LIN {X 0,Y 234.227,Z 351.546,A -85,B 0,C 180,E1 9411.137,E2 9411.137} C_VEL
LIN {X 0,Y 232.184,Z 350.426,A -85,B 0,C 180,E1 9404.231,E2 9404.231} C_VEL
LIN {X 0,Y 231.874,Z 350.167,A -85,B 0,C 180,E1 9397.903,E2 9397.903} C_VEL
LIN {X 0,Y 232.888,Z 350.916,A -85,B 0,C 180,E1 9391.006,E2 9391.006} C_VEL
LIN {X 0,Y 234.314,Z 351.747,A -85,B 0,C 180,E1 9386.888,E2 9386.888} C_VEL
LIN {X 0,Y 236.206,Z 355.562,A -85,B 0,C 180,E1 9382.033,E2 9382.033} C_VEL
LIN {X 0,Y 238.881,Z 357.916,A -85,B 0,C 180,E1 9377.787,E2 9377.787} C_VEL
LIN {X 0,Y 241.494,Z 361.984,A -85,B 0,C 180,E1 9374.013,E2 9374.013} C_VEL
LIN {X 0,Y 243.571,Z 364.124,A -85,B 0,C 180,E1 9371.6,E2 9371.6} C_VEL
LIN {X 0,Y 247.204,Z 368.916,A -85,B 0,C 180,E1 9367.74,E2 9367.74} C_VEL
LIN {X 0,Y 252.401,Z 375.828,A -85,B 0,C 180,E1 9363.074,E2 9363.074} C_VEL
LIN {X 0,Y 256.798,Z 381.754,A -85,B 0,C 180,E1 9359.662,E2 9359.662} C_VEL
LIN {X 0,Y 261.47,Z 388.445,A -85,B 0,C 180,E1 9356.385,E2 9356.385} C_VEL
LIN {X 0,Y 268.294,Z 399.263,A -85,B 0,C 180,E1 9352.072,E2 9352.072} C_VEL
LIN {X 0,Y 276.387,Z 412.565,A -85,B 0,C 180,E1 9347.608,E2 9347.608} C_VEL
LIN {X 0,Y 284.443,Z 426.777,A -85,B 0,C 180,E1 9343.665,E2 9343.665} C_VEL
LIN {X 0,Y 289.912,Z 436.98,A -85,B 0,C 180,E1 9341.23,E2 9341.23} C_VEL
LIN {X 0,Y 275.033,Z 547.244,A -85,B 0,C 180,E1 9338.255,E2 9338.255} C_VEL
LIN {X 0,Y 273.431,Z 554.838,A -85,B 0,C 180,E1 9338.207,E2 9338.207} C_VEL
LIN {X 0,Y 266.861,Z 574.928,A -85,B 0,C 180,E1 9338.675,E2 9338.675} C_VEL
LIN {X 0,Y 265.438,Z 581.426,A -85,B 0,C 180,E1 9338.599,E2 9338.599} C_VEL
LIN {X 0,Y 260.934,Z 605.989,A -85,B 0,C 180,E1 9337.701,E2 9337.701} C_VEL
LIN {X 0,Y 255.076,Z 629.268,A -85,B 0,C 180,E1 9336.611,E2 9336.611} C_VEL
LIN {X 0,Y 248.158,Z 651.869,A -85,B 0,C 180,E1 9335.198,E2 9335.198} C_VEL
LIN {X 0,Y 240.392,Z 673.643,A -85,B 0,C 180,E1 9333.405,E2 9333.405} C_VEL
LIN {X 0,Y 231.725,Z 694.834,A -85,B 0,C 180,E1 9331.147,E2 9331.147} C_VEL
LIN {X 0,Y 223.215,Z 713.542,A -85,B 0,C 180,E1 9328.611,E2 9328.611} C_VEL
LIN {X 0,Y 213.828,Z 732.446,A -85,B 0,C 180,E1 9325.378,E2 9325.378} C_VEL
LIN {X 0,Y 204.768,Z 749.485,A -85,B 0,C 180,E1 9321.671,E2 9321.671} C_VEL
LIN {X 0,Y 196.426,Z 764.496,A -85,B 0,C 180,E1 9317.563,E2 9317.563} C_VEL
LIN {X 0,Y 188.528,Z 778.313,A -85,B 0,C 180,E1 9312.749,E2 9312.749} C_VEL
LIN {X 0,Y 181.922,Z 790.051,A -85,B 0,C 180,E1 9307.59,E2 9307.59} C_VEL
LIN {X 0,Y 176.376,Z 800.61,A -85,B 0,C 180,E1 9301.746,E2 9301.746} C_VEL
LIN {X 0,Y 172.499,Z 809.062,A -85,B 0,C 180,E1 9295.764,E2 9295.764} C_VEL
LIN {X 0,Y 170.003,Z 816.157,A -85,B 0,C 180,E1 9289.226,E2 9289.226} C_VEL
LIN {X 0,Y 169.005,Z 821.281,A -85,B 0,C 180,E1 9282.988,E2 9282.988} C_VEL
LIN {X 0,Y 168.985,Z 824.538,A -85,B 0,C 180,E1 9277.134,E2 9277.134} C_VEL
LIN {X 0,Y 169.187,Z 826.21,A -85,B 0,C 180,E1 9272.368,E2 9272.368} C_VEL
LIN {X 0,Y 169.127,Z 826.898,A -85,B 0,C 180,E1 9267.964,E2 9267.964} C_VEL
LIN {X 0,Y 168.776,Z 826.725,A -85,B 0,C 180,E1 9262.85,E2 9262.85} C_VEL
LIN {X 0,Y 168.789,Z 825.056,A -85,B 0,C 180,E1 9255.941,E2 9255.941} C_VEL
LIN {X 0,Y 170.369,Z 821.696,A -85,B 0,C 180,E1 9248.659,E2 9248.659} C_VEL
LIN {X 0,Y 174.906,Z 815.918,A -85,B 0,C 180,E1 9240.339,E2 9240.339} C_VEL
LIN {X 0,Y 182.577,Z 808.466,A -85,B 0,C 180,E1 9232.561,E2 9232.561} C_VEL
LIN {X 0,Y 195.682,Z 797.535,A -85,B 0,C 180,E1 9224.325,E2 9224.325} C_VEL
LIN {X 0,Y 212.712,Z 784.952,A -85,B 0,C 180,E1 9217.399,E2 9217.399} C_VEL
LIN {X 0,Y 222.74,Z 778.057,A -85,B 0,C 180,E1 9214.369,E2 9214.369} C_VEL
LIN {X 0,Y 204.082,Z 786.443,A -85,B 0,C 180,E1 9207.742,E2 9207.742} C_VEL
LIN {X 0,Y 189.979,Z 792.578,A -85,B 0,C 180,E1 9200.33,E2 9200.33} C_VEL
LIN {X 0,Y 180.154,Z 796.526,A -85,B 0,C 180,E1 9192.505,E2 9192.505} C_VEL
LIN {X 0,Y 173.807,Z 798.607,A -85,B 0,C 180,E1 9184.293,E2 9184.293} C_VEL
LIN {X 0,Y 170.626,Z 798.921,A -85,B 0,C 180,E1 9176.645,E2 9176.645} C_VEL
LIN {X 0,Y 169.369,Z 797.944,A -85,B 0,C 180,E1 9170.147,E2 9170.147} C_VEL
LIN {X 0,Y 168.986,Z 795.971,A -85,B 0,C 180,E1 9163.859,E2 9163.859} C_VEL
LIN {X 0,Y 169.098,Z 792.896,A -85,B 0,C 180,E1 9157.769,E2 9157.769} C_VEL
LIN {X 0,Y 170.029,Z 788.306,A -85,B 0,C 180,E1 9151.177,E2 9151.177} C_VEL
LIN {X 0,Y 172.203,Z 782.022,A -85,B 0,C 180,E1 9144.512,E2 9144.512} C_VEL
LIN {X 0,Y 175.758,Z 774.235,A -85,B 0,C 180,E1 9138.183,E2 9138.183} C_VEL
LIN {X 0,Y 180.978,Z 764.462,A -85,B 0,C 180,E1 9131.954,E2 9131.954} C_VEL
LIN {X 0,Y 187.436,Z 753.199,A -85,B 0,C 180,E1 9126.311,E2 9126.311} C_VEL
LIN {X 0,Y 195.068,Z 740.016,A -85,B 0,C 180,E1 9121.141,E2 9121.141} C_VEL
LIN {X 0,Y 203.143,Z 725.828,A -85,B 0,C 180,E1 9116.72,E2 9116.72} C_VEL
LIN {X 0,Y 212.222,Z 709.143,A -85,B 0,C 180,E1 9112.58,E2 9112.58} C_VEL
LIN {X 0,Y 221.157,Z 691.592,A -85,B 0,C 180,E1 9109.124,E2 9109.124} C_VEL
LIN {X 0,Y 230.01,Z 672.581,A -85,B 0,C 180,E1 9106.135,E2 9106.135} C_VEL
LIN {X 0,Y 238.598,Z 651.957,A -85,B 0,C 180,E1 9103.559,E2 9103.559} C_VEL
LIN {X 0,Y 246.314,Z 630.844,A -85,B 0,C 180,E1 9101.475,E2 9101.475} C_VEL
LIN {X 0,Y 253.119,Z 609.216,A -85,B 0,C 180,E1 9099.782,E2 9099.782} C_VEL
LIN {X 0,Y 259.157,Z 586.244,A -85,B 0,C 180,E1 9098.374,E2 9098.374} C_VEL
LIN {X 0,Y 264.081,Z 562.955,A -85,B 0,C 180,E1 9097.296,E2 9097.296} C_VEL
LIN {X 0,Y 267.959,Z 538.7,A -85,B 0,C 180,E1 9096.486,E2 9096.486} C_VEL
LIN {X 0,Y 282.577,Z 431.743,A -85,B 0,C 180,E1 9093.574,E2 9093.574} C_VEL
LIN {X 0,Y 274.363,Z 418.564,A -85,B 0,C 180,E1 9089.741,E2 9089.741} C_VEL
LIN {X 0,Y 266.819,Z 407.093,A -85,B 0,C 180,E1 9085.758,E2 9085.758} C_VEL
LIN {X 0,Y 259.677,Z 396.52,A -85,B 0,C 180,E1 9081.434,E2 9081.434} C_VEL
LIN {X 0,Y 252.796,Z 386.86,A -85,B 0,C 180,E1 9076.631,E2 9076.631} C_VEL
LIN {X 0,Y 248.348,Z 380.97,A -85,B 0,C 180,E1 9073.032,E2 9073.032} C_VEL
LIN {X 0,Y 244.808,Z 376.083,A -85,B 0,C 180,E1 9069.689,E2 9069.689} C_VEL
LIN {X 0,Y 240.82,Z 370.808,A -85,B 0,C 180,E1 9065.393,E2 9065.393} C_VEL
LIN {X 0,Y 237.474,Z 366.554,A -85,B 0,C 180,E1 9061.043,E2 9061.043} C_VEL
LIN {X 0,Y 236.712,Z 365.222,A -85,B 0,C 180,E1 9059.828,E2 9059.828} C_VEL
LIN {X 0,Y 233.699,Z 362.264,A -85,B 0,C 180,E1 9054.723,E2 9054.723} C_VEL
LIN {X 0,Y 232.484,Z 359.353,A -85,B 0,C 180,E1 9051.108,E2 9051.108} C_VEL
LIN {X 0,Y 230.463,Z 358.25,A -85,B 0,C 180,E1 9044.292,E2 9044.292} C_VEL
LIN {X 0,Y 230.127,Z 357.958,A -85,B 0,C 180,E1 9038.089,E2 9038.089} C_VEL
LIN {X 0,Y 231.138,Z 358.717,A -85,B 0,C 180,E1 9031.079,E2 9031.079} C_VEL
LIN {X 0,Y 232.525,Z 359.644,A -85,B 0,C 180,E1 9026.988,E2 9026.988} C_VEL
LIN {X 0,Y 234.468,Z 363.42,A -85,B 0,C 180,E1 9022.037,E2 9022.037} C_VEL
LIN {X 0,Y 236.948,Z 365.661,A -85,B 0,C 180,E1 9018.064,E2 9018.064} C_VEL
LIN {X 0,Y 239.763,Z 369.906,A -85,B 0,C 180,E1 9013.993,E2 9013.993} C_VEL
LIN {X 0,Y 241.496,Z 371.753,A -85,B 0,C 180,E1 9011.944,E2 9011.944} C_VEL
LIN {X 0,Y 245.087,Z 376.49,A -85,B 0,C 180,E1 9008.088,E2 9008.088} C_VEL
LIN {X 0,Y 250.177,Z 383.4,A -85,B 0,C 180,E1 9003.434,E2 9003.434} C_VEL
LIN {X 0,Y 254.304,Z 389.018,A -85,B 0,C 180,E1 9000.166,E2 9000.166} C_VEL
LIN {X 0,Y 258.815,Z 395.549,A -85,B 0,C 180,E1 8996.952,E2 8996.952} C_VEL
LIN {X 0,Y 266.166,Z 407.353,A -85,B 0,C 180,E1 8992.225,E2 8992.225} C_VEL
LIN {X 0,Y 274.005,Z 420.688,A -85,B 0,C 180,E1 8987.832,E2 8987.832} C_VEL
LIN {X 0,Y 282.179,Z 435.229,A -85,B 0,C 180,E1 8983.807,E2 8983.807} C_VEL
LIN {X 0,Y 285.025,Z 440.843,A -85,B 0,C 180,E1 8982.469,E2 8982.469} C_VEL
LIN {X 0,Y 265.438,Z 581.426,A -85,B 0,C 180,E1 8978.599,E2 8978.599} C_VEL
LIN {X 0,Y 263.629,Z 588.969,A -85,B 0,C 180,E1 8978.531,E2 8978.531} C_VEL
LIN {X 0,Y 255.789,Z 608.692,A -85,B 0,C 180,E1 8978.847,E2 8978.847} C_VEL
LIN {X 0,Y 253.732,Z 615.005,A -85,B 0,C 180,E1 8978.695,E2 8978.695} C_VEL
LIN {X 0,Y 247.281,Z 637.887,A -85,B 0,C 180,E1 8977.498,E2 8977.498} C_VEL
LIN {X 0,Y 239.575,Z 660.767,A -85,B 0,C 180,E1 8975.882,E2 8975.882} C_VEL
LIN {X 0,Y 231.448,Z 681.602,A -85,B 0,C 180,E1 8973.962,E2 8973.962} C_VEL
LIN {X 0,Y 222.706,Z 701.487,A -85,B 0,C 180,E1 8971.631,E2 8971.631} C_VEL
LIN {X 0,Y 213.051,Z 721.326,A -85,B 0,C 180,E1 8968.658,E2 8968.658} C_VEL
LIN {X 0,Y 203.867,Z 738.763,A -85,B 0,C 180,E1 8965.322,E2 8965.322} C_VEL
LIN {X 0,Y 194.615,Z 755.189,A -85,B 0,C 180,E1 8961.339,E2 8961.339} C_VEL
LIN {X 0,Y 185.72,Z 770.316,A -85,B 0,C 180,E1 8956.613,E2 8956.613} C_VEL
LIN {X 0,Y 178.084,Z 783.164,A -85,B 0,C 180,E1 8951.487,E2 8951.487} C_VEL
LIN {X 0,Y 171.499,Z 794.656,A -85,B 0,C 180,E1 8945.658,E2 8945.658} C_VEL
LIN {X 0,Y 166.516,Z 804.244,A -85,B 0,C 180,E1 8939.457,E2 8939.457} C_VEL
LIN {X 0,Y 163.225,Z 811.808,A -85,B 0,C 180,E1 8933.078,E2 8933.078} C_VEL
LIN {X 0,Y 161.396,Z 818.085,A -85,B 0,C 180,E1 8926.183,E2 8926.183} C_VEL
LIN {X 0,Y 160.973,Z 822.135,A -85,B 0,C 180,E1 8920.012,E2 8920.012} C_VEL
LIN {X 0,Y 161.189,Z 824.814,A -85,B 0,C 180,E1 8913.909,E2 8913.909} C_VEL
LIN {X 0,Y 161.231,Z 825.868,A -85,B 0,C 180,E1 8908.93,E2 8908.93} C_VEL
LIN {X 0,Y 160.87,Z 825.957,A -85,B 0,C 180,E1 8903.573,E2 8903.573} C_VEL
LIN {X 0,Y 160.714,Z 824.926,A -85,B 0,C 180,E1 8897.42,E2 8897.42} C_VEL
LIN {X 0,Y 162.078,Z 822.073,A -85,B 0,C 180,E1 8889.409,E2 8889.409} C_VEL
LIN {X 0,Y 166.066,Z 817.315,A -85,B 0,C 180,E1 8881.202,E2 8881.202} C_VEL
LIN {X 0,Y 174.264,Z 809.955,A -85,B 0,C 180,E1 8872.358,E2 8872.358} C_VEL
LIN {X 0,Y 187.354,Z 800.105,A -85,B 0,C 180,E1 8863.904,E2 8863.904} C_VEL
LIN {X 0,Y 205.303,Z 788.102,A -85,B 0,C 180,E1 8856.524,E2 8856.524} C_VEL
LIN {X 0,Y 212.518,Z 783.476,A -85,B 0,C 180,E1 8854.213,E2 8854.213} C_VEL
LIN {X 0,Y 194.093,Z 790.664,A -85,B 0,C 180,E1 8847.293,E2 8847.293} C_VEL
LIN {X 0,Y 179.763,Z 795.903,A -85,B 0,C 180,E1 8839.161,E2 8839.161} C_VEL
LIN {X 0,Y 170.394,Z 798.849,A -85,B 0,C 180,E1 8830.827,E2 8830.827} C_VEL
LIN {X 0,Y 164.969,Z 799.982,A -85,B 0,C 180,E1 8822.784,E2 8822.784} C_VEL
LIN {X 0,Y 162.228,Z 799.597,A -85,B 0,C 180,E1 8815.055,E2 8815.055} C_VEL
LIN {X 0,Y 161.179,Z 797.931,A -85,B 0,C 180,E1 8807.829,E2 8807.829} C_VEL
LIN {X 0,Y 160.981,Z 795.623,A -85,B 0,C 180,E1 8801.867,E2 8801.867} C_VEL
LIN {X 0,Y 161.361,Z 791.817,A -85,B 0,C 180,E1 8795.086,E2 8795.086} C_VEL
LIN {X 0,Y 162.698,Z 786.804,A -85,B 0,C 180,E1 8788.515,E2 8788.515} C_VEL
LIN {X 0,Y 165.56,Z 779.753,A -85,B 0,C 180,E1 8781.542,E2 8781.542} C_VEL
LIN {X 0,Y 170.173,Z 770.773,A -85,B 0,C 180,E1 8774.696,E2 8774.696} C_VEL
LIN {X 0,Y 176.24,Z 760.286,A -85,B 0,C 180,E1 8768.481,E2 8768.481} C_VEL
LIN {X 0,Y 183.761,Z 747.753,A -85,B 0,C 180,E1 8762.717,E2 8762.717} C_VEL
LIN {X 0,Y 192.036,Z 733.936,A -85,B 0,C 180,E1 8757.745,E2 8757.745} C_VEL
LIN {X 0,Y 200.939,Z 718.552,A -85,B 0,C 180,E1 8753.369,E2 8753.369} C_VEL
LIN {X 0,Y 210.109,Z 701.775,A -85,B 0,C 180,E1 8749.585,E2 8749.585} C_VEL
LIN {X 0,Y 219.291,Z 683.595,A -85,B 0,C 180,E1 8746.323,E2 8746.323} C_VEL
LIN {X 0,Y 228.281,Z 663.897,A -85,B 0,C 180,E1 8743.525,E2 8743.525} C_VEL
LIN {X 0,Y 236.572,Z 643.38,A -85,B 0,C 180,E1 8741.213,E2 8741.213} C_VEL
LIN {X 0,Y 244.149,Z 621.904,A -85,B 0,C 180,E1 8739.29,E2 8739.29} C_VEL
LIN {X 0,Y 250.933,Z 599.279,A -85,B 0,C 180,E1 8737.7,E2 8737.7} C_VEL
LIN {X 0,Y 256.726,Z 575.762,A -85,B 0,C 180,E1 8736.434,E2 8736.434} C_VEL
LIN {X 0,Y 261.268,Z 552.258,A -85,B 0,C 180,E1 8735.497,E2 8735.497} C_VEL
LIN {X 0,Y 277.761,Z 435.917,A -85,B 0,C 180,E1 8732.271,E2 8732.271} C_VEL
LIN {X 0,Y 270.034,Z 423.47,A -85,B 0,C 180,E1 8728.504,E2 8728.504} C_VEL
LIN {X 0,Y 262.754,Z 412.255,A -85,B 0,C 180,E1 8724.489,E2 8724.489} C_VEL
LIN {X 0,Y 256.44,Z 402.941,A -85,B 0,C 180,E1 8720.529,E2 8720.529} C_VEL
LIN {X 0,Y 251.756,Z 396.305,A -85,B 0,C 180,E1 8717.21,E2 8717.21} C_VEL
LIN {X 0,Y 246.641,Z 389.023,A -85,B 0,C 180,E1 8713.066,E2 8713.066} C_VEL
LIN {X 0,Y 242.563,Z 383.544,A -85,B 0,C 180,E1 8709.24,E2 8709.24} C_VEL
LIN {X 0,Y 238.714,Z 378.371,A -85,B 0,C 180,E1 8704.976,E2 8704.976} C_VEL
LIN {X 0,Y 235.286,Z 373.743,A -85,B 0,C 180,E1 8700.329,E2 8700.329} C_VEL
LIN {X 0,Y 234.542,Z 372.775,A -85,B 0,C 180,E1 8699.235,E2 8699.235} C_VEL
LIN {X 0,Y 231.803,Z 369.92,A -85,B 0,C 180,E1 8694.391,E2 8694.391} C_VEL
LIN {X 0,Y 230.573,Z 367.105,A -85,B 0,C 180,E1 8690.723,E2 8690.723} C_VEL
LIN {X 0,Y 228.698,Z 366.025,A -85,B 0,C 180,E1 8684.032,E2 8684.032} C_VEL
LIN {X 0,Y 228.44,Z 365.833,A -85,B 0,C 180,E1 8677.468,E2 8677.468} C_VEL
LIN {X 0,Y 229.527,Z 366.593,A -85,B 0,C 180,E1 8670.637,E2 8670.637} C_VEL
LIN {X 0,Y 230.701,Z 367.411,A -85,B 0,C 180,E1 8667.218,E2 8667.218} C_VEL
LIN {X 0,Y 232.632,Z 371.172,A -85,B 0,C 180,E1 8662.22,E2 8662.22} C_VEL
LIN {X 0,Y 235.01,Z 373.395,A -85,B 0,C 180,E1 8658.347,E2 8658.347} C_VEL
LIN {X 0,Y 238.017,Z 377.803,A -85,B 0,C 180,E1 8653.993,E2 8653.993} C_VEL
LIN {X 0,Y 239.519,Z 379.541,A -85,B 0,C 180,E1 8652.178,E2 8652.178} C_VEL
LIN {X 0,Y 243.727,Z 385.197,A -85,B 0,C 180,E1 8647.659,E2 8647.659} C_VEL
LIN {X 0,Y 247.988,Z 391.039,A -85,B 0,C 180,E1 8643.753,E2 8643.753} C_VEL
LIN {X 0,Y 251.829,Z 396.283,A -85,B 0,C 180,E1 8640.679,E2 8640.679} C_VEL
LIN {X 0,Y 256.198,Z 402.745,A -85,B 0,C 180,E1 8637.483,E2 8637.483} C_VEL
LIN {X 0,Y 263.347,Z 414.383,A -85,B 0,C 180,E1 8632.8,E2 8632.8} C_VEL
LIN {X 0,Y 271.117,Z 427.821,A -85,B 0,C 180,E1 8628.349,E2 8628.349} C_VEL
LIN {X 0,Y 278.913,Z 441.987,A -85,B 0,C 180,E1 8624.401,E2 8624.401} C_VEL
LIN {X 0,Y 280.247,Z 444.727,A -85,B 0,C 180,E1 8623.748,E2 8623.748} C_VEL
LIN {X 0,Y 259.573,Z 587.76,A -85,B 0,C 180,E1 8619.781,E2 8619.781} C_VEL
LIN {X 0,Y 254.518,Z 611.914,A -85,B 0,C 180,E1 8618.833,E2 8618.833} C_VEL
LIN {X 0,Y 253.732,Z 615.005,A -85,B 0,C 180,E1 8618.695,E2 8618.695} C_VEL
LIN {X 0,Y 251.096,Z 622.267,A -85,B 0,C 180,E1 8618.542,E2 8618.542} C_VEL
LIN {X 0,Y 241.864,Z 640.153,A -85,B 0,C 180,E1 8618.605,E2 8618.605} C_VEL
LIN {X 0,Y 238.932,Z 647.239,A -85,B 0,C 180,E1 8618.3,E2 8618.3} C_VEL
LIN {X 0,Y 230.958,Z 668.879,A -85,B 0,C 180,E1 8616.597,E2 8616.597} C_VEL
LIN {X 0,Y 222.143,Z 689.76,A -85,B 0,C 180,E1 8614.474,E2 8614.474} C_VEL
LIN {X 0,Y 212.642,Z 709.884,A -85,B 0,C 180,E1 8611.834,E2 8611.834} C_VEL
LIN {X 0,Y 203.302,Z 727.849,A -85,B 0,C 180,E1 8608.836,E2 8608.836} C_VEL
LIN {X 0,Y 193.345,Z 745.554,A -85,B 0,C 180,E1 8605.045,E2 8605.045} C_VEL
LIN {X 0,Y 183.748,Z 761.589,A -85,B 0,C 180,E1 8600.59,E2 8600.59} C_VEL
LIN {X 0,Y 175.521,Z 774.886,A -85,B 0,C 180,E1 8595.865,E2 8595.865} C_VEL
LIN {X 0,Y 168.101,Z 786.996,A -85,B 0,C 180,E1 8590.411,E2 8590.411} C_VEL
LIN {X 0,Y 161.684,Z 798.017,A -85,B 0,C 180,E1 8584.032,E2 8584.032} C_VEL
LIN {X 0,Y 157.086,Z 806.918,A -85,B 0,C 180,E1 8577.272,E2 8577.272} C_VEL
LIN {X 0,Y 154.193,Z 814.321,A -85,B 0,C 180,E1 8569.897,E2 8569.897} C_VEL
LIN {X 0,Y 153.095,Z 819.596,A -85,B 0,C 180,E1 8562.826,E2 8562.826} C_VEL
LIN {X 0,Y 153.143,Z 822.832,A -85,B 0,C 180,E1 8556.369,E2 8556.369} C_VEL
LIN {X 0,Y 153.333,Z 824.367,A -85,B 0,C 180,E1 8551.491,E2 8551.491} C_VEL
LIN {X 0,Y 153.181,Z 825.021,A -85,B 0,C 180,E1 8547.003,E2 8547.003} C_VEL
LIN {X 0,Y 152.764,Z 824.882,A -85,B 0,C 180,E1 8541.255,E2 8541.255} C_VEL
LIN {X 0,Y 153.021,Z 823.484,A -85,B 0,C 180,E1 8534.068,E2 8534.068} C_VEL
LIN {X 0,Y 155.573,Z 820.05,A -85,B 0,C 180,E1 8525.304,E2 8525.304} C_VEL
LIN {X 0,Y 161.418,Z 814.856,A -85,B 0,C 180,E1 8516.541,E2 8516.541} C_VEL
LIN {X 0,Y 172.449,Z 806.769,A -85,B 0,C 180,E1 8507.28,E2 8507.28} C_VEL
LIN {X 0,Y 188.846,Z 796.295,A -85,B 0,C 180,E1 8498.891,E2 8498.891} C_VEL
LIN {X 0,Y 202.423,Z 788.339,A -85,B 0,C 180,E1 8494.12,E2 8494.12} C_VEL
LIN {X 0,Y 184.041,Z 794.454,A -85,B 0,C 180,E1 8486.807,E2 8486.807} C_VEL
LIN {X 0,Y 170.344,Z 798.54,A -85,B 0,C 180,E1 8478.484,E2 8478.484} C_VEL
LIN {X 0,Y 161.314,Z 800.652,A -85,B 0,C 180,E1 8469.747,E2 8469.747} C_VEL
LIN {X 0,Y 156.024,Z 801.021,A -85,B 0,C 180,E1 8460.739,E2 8460.739} C_VEL
LIN {X 0,Y 153.806,Z 799.883,A -85,B 0,C 180,E1 8452.91,E2 8452.91} C_VEL
LIN {X 0,Y 153.085,Z 797.762,A -85,B 0,C 180,E1 8445.635,E2 8445.635} C_VEL
LIN {X 0,Y 153.06,Z 794.662,A -85,B 0,C 180,E1 8438.95,E2 8438.95} C_VEL
LIN {X 0,Y 153.833,Z 790.405,A -85,B 0,C 180,E1 8432.104,E2 8432.104} C_VEL
LIN {X 0,Y 155.954,Z 784.185,A -85,B 0,C 180,E1 8424.766,E2 8424.766} C_VEL
LIN {X 0,Y 159.832,Z 776.159,A -85,B 0,C 180,E1 8417.506,E2 8417.506} C_VEL
LIN {X 0,Y 165.354,Z 766.551,A -85,B 0,C 180,E1 8410.776,E2 8410.776} C_VEL
LIN {X 0,Y 172.417,Z 755.099,A -85,B 0,C 180,E1 8404.576,E2 8404.576} C_VEL
LIN {X 0,Y 180.42,Z 742.284,A -85,B 0,C 180,E1 8399.191,E2 8399.191} C_VEL
LIN {X 0,Y 189.512,Z 727.46,A -85,B 0,C 180,E1 8394.304,E2 8394.304} C_VEL
LIN {X 0,Y 199.052,Z 711.11,A -85,B 0,C 180,E1 8390.077,E2 8390.077} C_VEL
LIN {X 0,Y 208.562,Z 693.631,A -85,B 0,C 180,E1 8386.52,E2 8386.52} C_VEL
LIN {X 0,Y 217.949,Z 674.718,A -85,B 0,C 180,E1 8383.473,E2 8383.473} C_VEL
LIN {X 0,Y 227.019,Z 654.18,A -85,B 0,C 180,E1 8380.865,E2 8380.865} C_VEL
LIN {X 0,Y 235.147,Z 633.27,A -85,B 0,C 180,E1 8378.769,E2 8378.769} C_VEL
LIN {X 0,Y 242.435,Z 611.542,A -85,B 0,C 180,E1 8377.048,E2 8377.048} C_VEL
LIN {X 0,Y 248.904,Z 588.492,A -85,B 0,C 180,E1 8375.625,E2 8375.625} C_VEL
LIN {X 0,Y 254.149,Z 565.347,A -85,B 0,C 180,E1 8374.539,E2 8374.539} C_VEL
LIN {X 0,Y 258.358,Z 540.834,A -85,B 0,C 180,E1 8373.709,E2 8373.709} C_VEL
LIN {X 0,Y 273.067,Z 440.173,A -85,B 0,C 180,E1 8370.972,E2 8370.972} C_VEL
LIN {X 0,Y 265.083,Z 427.25,A -85,B 0,C 180,E1 8366.867,E2 8366.867} C_VEL
LIN {X 0,Y 257.223,Z 415.133,A -85,B 0,C 180,E1 8362.245,E2 8362.245} C_VEL
LIN {X 0,Y 250.737,Z 405.62,A -85,B 0,C 180,E1 8357.801,E2 8357.801} C_VEL
LIN {X 0,Y 246.647,Z 399.831,A -85,B 0,C 180,E1 8354.564,E2 8354.564} C_VEL
LIN {X 0,Y 243.563,Z 395.565,A -85,B 0,C 180,E1 8351.947,E2 8351.947} C_VEL
LIN {X 0,Y 240.287,Z 390.964,A -85,B 0,C 180,E1 8348.75,E2 8348.75} C_VEL
LIN {X 0,Y 236.695,Z 386.016,A -85,B 0,C 180,E1 8344.677,E2 8344.677} C_VEL
LIN {X 0,Y 233.279,Z 381.357,A -85,B 0,C 180,E1 8339.964,E2 8339.964} C_VEL
LIN {X 0,Y 232.398,Z 380.326,A -85,B 0,C 180,E1 8338.632,E2 8338.632} C_VEL
LIN {X 0,Y 229.889,Z 377.529,A -85,B 0,C 180,E1 8333.988,E2 8333.988} C_VEL
LIN {X 0,Y 228.663,Z 374.848,A -85,B 0,C 180,E1 8330.309,E2 8330.309} C_VEL
LIN {X 0,Y 226.933,Z 373.799,A -85,B 0,C 180,E1 8323.737,E2 8323.737} C_VEL
LIN {X 0,Y 226.708,Z 373.655,A -85,B 0,C 180,E1 8317.167,E2 8317.167} C_VEL
LIN {X 0,Y 227.894,Z 374.463,A -85,B 0,C 180,E1 8310.297,E2 8310.297} C_VEL
LIN {X 0,Y 228.881,Z 375.175,A -85,B 0,C 180,E1 8307.453,E2 8307.453} C_VEL
LIN {X 0,Y 230.942,Z 379.096,A -85,B 0,C 180,E1 8302.111,E2 8302.111} C_VEL
LIN {X 0,Y 233.105,Z 381.187,A -85,B 0,C 180,E1 8298.58,E2 8298.58} C_VEL
LIN {X 0,Y 236.306,Z 385.723,A -85,B 0,C 180,E1 8293.952,E2 8293.952} C_VEL
LIN {X 0,Y 237.55,Z 387.349,A -85,B 0,C 180,E1 8292.392,E2 8292.392} C_VEL
LIN {X 0,Y 241.612,Z 392.872,A -85,B 0,C 180,E1 8287.965,E2 8287.965} C_VEL
LIN {X 0,Y 245.624,Z 398.394,A -85,B 0,C 180,E1 8284.239,E2 8284.239} C_VEL
LIN {X 0,Y 249.652,Z 403.982,A -85,B 0,C 180,E1 8280.972,E2 8280.972} C_VEL
LIN {X 0,Y 253.793,Z 410.332,A -85,B 0,C 180,E1 8277.852,E2 8277.852} C_VEL
LIN {X 0,Y 260.366,Z 421.222,A -85,B 0,C 180,E1 8273.437,E2 8273.437} C_VEL
LIN {X 0,Y 267.867,Z 434.408,A -85,B 0,C 180,E1 8269.023,E2 8269.023} C_VEL
LIN {X 0,Y 275.28,Z 448.097,A -85,B 0,C 180,E1 8265.161,E2 8265.161} C_VEL
LIN {X 0,Y 275.416,Z 449.006,A -85,B 0,C 180,E1 8265.044,E2 8265.044} C_VEL
LIN {X 0,Y 254.8,Z 587.13,A -85,B 0,C 180,E1 8261.215,E2 8261.215} C_VEL
LIN {X 0,Y 249.61,Z 611.365,A -85,B 0,C 180,E1 8260.268,E2 8260.268} C_VEL
LIN {X 0,Y 243.163,Z 634.159,A -85,B 0,C 180,E1 8259.127,E2 8259.127} C_VEL
LIN {X 0,Y 238.932,Z 647.239,A -85,B 0,C 180,E1 8258.3,E2 8258.3} C_VEL
LIN {X 0,Y 235.843,Z 654.254,A -85,B 0,C 180,E1 8257.991,E2 8257.991} C_VEL
LIN {X 0,Y 224.656,Z 672.298,A -85,B 0,C 180,E1 8257.629,E2 8257.629} C_VEL
LIN {X 0,Y 221.692,Z 677.98,A -85,B 0,C 180,E1 8257.202,E2 8257.202} C_VEL
LIN {X 0,Y 212.126,Z 698.839,A -85,B 0,C 180,E1 8254.815,E2 8254.815} C_VEL
LIN {X 0,Y 202.379,Z 717.909,A -85,B 0,C 180,E1 8252.004,E2 8252.004} C_VEL
LIN {X 0,Y 192.218,Z 736.122,A -85,B 0,C 180,E1 8248.541,E2 8248.541} C_VEL
LIN {X 0,Y 182.04,Z 752.974,A -85,B 0,C 180,E1 8244.373,E2 8244.373} C_VEL
LIN {X 0,Y 172.892,Z 767.388,A -85,B 0,C 180,E1 8239.757,E2 8239.757} C_VEL
LIN {X 0,Y 163.982,Z 781.203,A -85,B 0,C 180,E1 8234.03,E2 8234.03} C_VEL
LIN {X 0,Y 156.7,Z 792.79,A -85,B 0,C 180,E1 8227.769,E2 8227.769} C_VEL
LIN {X 0,Y 151.181,Z 802.367,A -85,B 0,C 180,E1 8221.051,E2 8221.051} C_VEL
LIN {X 0,Y 147.496,Z 810.036,A -85,B 0,C 180,E1 8213.995,E2 8213.995} C_VEL
LIN {X 0,Y 145.498,Z 816.349,A -85,B 0,C 180,E1 8206.36,E2 8206.36} C_VEL
LIN {X 0,Y 145.097,Z 820.384,A -85,B 0,C 180,E1 8199.515,E2 8199.515} C_VEL
LIN {X 0,Y 145.341,Z 822.773,A -85,B 0,C 180,E1 8193.546,E2 8193.546} C_VEL
LIN {X 0,Y 145.334,Z 823.878,A -85,B 0,C 180,E1 8188.419,E2 8188.419} C_VEL
LIN {X 0,Y 144.873,Z 824.147,A -85,B 0,C 180,E1 8182.461,E2 8182.461} C_VEL
LIN {X 0,Y 144.993,Z 822.997,A -85,B 0,C 180,E1 8174.395,E2 8174.395} C_VEL
LIN {X 0,Y 147.359,Z 820.238,A -85,B 0,C 180,E1 8165.546,E2 8165.546} C_VEL
LIN {X 0,Y 153.546,Z 815.261,A -85,B 0,C 180,E1 8155.939,E2 8155.939} C_VEL
LIN {X 0,Y 164.985,Z 807.884,A -85,B 0,C 180,E1 8146.297,E2 8146.297} C_VEL
LIN {X 0,Y 182.58,Z 797.928,A -85,B 0,C 180,E1 8137.429,E2 8137.429} C_VEL
LIN {X 0,Y 192.057,Z 792.801,A -85,B 0,C 180,E1 8133.958,E2 8133.958} C_VEL
LIN {X 0,Y 173.939,Z 797.814,A -85,B 0,C 180,E1 8126.276,E2 8126.276} C_VEL
LIN {X 0,Y 160.489,Z 800.922,A -85,B 0,C 180,E1 8117.405,E2 8117.405} C_VEL
LIN {X 0,Y 151.821,Z 802.157,A -85,B 0,C 180,E1 8107.954,E2 8107.954} C_VEL
LIN {X 0,Y 147.295,Z 801.636,A -85,B 0,C 180,E1 8098.838,E2 8098.838} C_VEL
LIN {X 0,Y 145.466,Z 799.858,A -85,B 0,C 180,E1 8090.51,E2 8090.51} C_VEL
LIN {X 0,Y 145.037,Z 797.551,A -85,B 0,C 180,E1 8083.999,E2 8083.999} C_VEL
LIN {X 0,Y 145.201,Z 794.069,A -85,B 0,C 180,E1 8076.896,E2 8076.896} C_VEL
LIN {X 0,Y 146.41,Z 788.965,A -85,B 0,C 180,E1 8069.376,E2 8069.376} C_VEL
LIN {X 0,Y 149.335,Z 781.919,A -85,B 0,C 180,E1 8061.496,E2 8061.496} C_VEL
LIN {X 0,Y 153.842,Z 773.65,A -85,B 0,C 180,E1 8054.372,E2 8054.372} C_VEL
LIN {X 0,Y 160.18,Z 763.329,A -85,B 0,C 180,E1 8047.567,E2 8047.567} C_VEL
LIN {X 0,Y 168.035,Z 751.2,A -85,B 0,C 180,E1 8041.376,E2 8041.376} C_VEL
LIN {X 0,Y 176.86,Z 737.612,A -85,B 0,C 180,E1 8036,E2 8036} C_VEL
LIN {X 0,Y 186.16,Z 722.829,A -85,B 0,C 180,E1 8031.424,E2 8031.424} C_VEL
LIN {X 0,Y 196.301,Z 705.692,A -85,B 0,C 180,E1 8027.289,E2 8027.289} C_VEL
LIN {X 0,Y 206.215,Z 687.358,A -85,B 0,C 180,E1 8023.844,E2 8023.844} C_VEL
LIN {X 0,Y 215.388,Z 668.645,A -85,B 0,C 180,E1 8021.068,E2 8021.068} C_VEL
LIN {X 0,Y 224.487,Z 647.85,A -85,B 0,C 180,E1 8018.624,E2 8018.624} C_VEL
LIN {X 0,Y 232.542,Z 626.773,A -85,B 0,C 180,E1 8016.669,E2 8016.669} C_VEL
LIN {X 0,Y 239.658,Z 605.026,A -85,B 0,C 180,E1 8015.077,E2 8015.077} C_VEL
LIN {X 0,Y 246.095,Z 581.122,A -85,B 0,C 180,E1 8013.729,E2 8013.729} C_VEL
LIN {X 0,Y 251.379,Z 556.029,A -85,B 0,C 180,E1 8012.696,E2 8012.696} C_VEL
LIN {X 0,Y 268.336,Z 444.458,A -85,B 0,C 180,E1 8009.629,E2 8009.629} C_VEL
LIN {X 0,Y 261.871,Z 433.854,A -85,B 0,C 180,E1 8006.171,E2 8006.171} C_VEL
LIN {X 0,Y 255.131,Z 423.302,A -85,B 0,C 180,E1 8002.119,E2 8002.119} C_VEL
LIN {X 0,Y 249.532,Z 414.854,A -85,B 0,C 180,E1 7998.269,E2 7998.269} C_VEL
LIN {X 0,Y 244.677,Z 407.757,A -85,B 0,C 180,E1 7994.444,E2 7994.444} C_VEL
LIN {X 0,Y 241.185,Z 402.852,A -85,B 0,C 180,E1 7991.387,E2 7991.387} C_VEL
LIN {X 0,Y 237.975,Z 398.321,A -85,B 0,C 180,E1 7988.195,E2 7988.195} C_VEL
LIN {X 0,Y 234.46,Z 393.467,A -85,B 0,C 180,E1 7984.123,E2 7984.123} C_VEL
LIN {X 0,Y 231.208,Z 388.814,A -85,B 0,C 180,E1 7979.464,E2 7979.464} C_VEL
LIN {X 0,Y 227.965,Z 385.097,A -85,B 0,C 180,E1 7973.525,E2 7973.525} C_VEL
LIN {X 0,Y 226.932,Z 382.659,A -85,B 0,C 180,E1 7970.297,E2 7970.297} C_VEL
LIN {X 0,Y 225.194,Z 381.602,A -85,B 0,C 180,E1 7963.642,E2 7963.642} C_VEL
LIN {X 0,Y 224.976,Z 381.464,A -85,B 0,C 180,E1 7957.182,E2 7957.182} C_VEL
LIN {X 0,Y 226.171,Z 382.284,A -85,B 0,C 180,E1 7950.258,E2 7950.258} C_VEL
LIN {X 0,Y 227.057,Z 382.894,A -85,B 0,C 180,E1 7947.741,E2 7947.741} C_VEL
LIN {X 0,Y 229.099,Z 386.843,A -85,B 0,C 180,E1 7942.305,E2 7942.305} C_VEL
LIN {X 0,Y 231.151,Z 388.841,A -85,B 0,C 180,E1 7938.926,E2 7938.926} C_VEL
LIN {X 0,Y 234.476,Z 393.522,A -85,B 0,C 180,E1 7934.064,E2 7934.064} C_VEL
LIN {X 0,Y 235.878,Z 395.642,A -85,B 0,C 180,E1 7932.233,E2 7932.233} C_VEL
LIN {X 0,Y 239.276,Z 400.151,A -85,B 0,C 180,E1 7928.527,E2 7928.527} C_VEL
LIN {X 0,Y 243.365,Z 405.888,A -85,B 0,C 180,E1 7924.651,E2 7924.651} C_VEL
LIN {X 0,Y 247.289,Z 411.438,A -85,B 0,C 180,E1 7921.387,E2 7921.387} C_VEL
LIN {X 0,Y 251.373,Z 417.893,A -85,B 0,C 180,E1 7918.23,E2 7918.23} C_VEL
LIN {X 0,Y 257.649,Z 428.521,A -85,B 0,C 180,E1 7913.927,E2 7913.927} C_VEL
LIN {X 0,Y 264.551,Z 440.822,A -85,B 0,C 180,E1 7909.765,E2 7909.765} C_VEL
LIN {X 0,Y 270.795,Z 452.583,A -85,B 0,C 180,E1 7906.397,E2 7906.397} C_VEL
LIN {X 0,Y 250.074,Z 587.129,A -85,B 0,C 180,E1 7902.68,E2 7902.68} C_VEL
LIN {X 0,Y 244.773,Z 611.188,A -85,B 0,C 180,E1 7901.745,E2 7901.745} C_VEL
LIN {X 0,Y 238.012,Z 634.438,A -85,B 0,C 180,E1 7900.586,E2 7900.586} C_VEL
LIN {X 0,Y 230.56,Z 655.892,A -85,B 0,C 180,E1 7899.147,E2 7899.147} C_VEL
LIN {X 0,Y 221.692,Z 677.98,A -85,B 0,C 180,E1 7897.202,E2 7897.202} C_VEL
LIN {X 0,Y 218.118,Z 684.605,A -85,B 0,C 180,E1 7896.7,E2 7896.7} C_VEL
LIN {X 0,Y 205.581,Z 701.473,A -85,B 0,C 180,E1 7895.844,E2 7895.844} C_VEL
LIN {X 0,Y 202.246,Z 706.801,A -85,B 0,C 180,E1 7895.226,E2 7895.226} C_VEL
LIN {X 0,Y 191.765,Z 725.887,A -85,B 0,C 180,E1 7892.061,E2 7892.061} C_VEL
LIN {X 0,Y 181.132,Z 743.584,A -85,B 0,C 180,E1 7888.214,E2 7888.214} C_VEL
LIN {X 0,Y 171.058,Z 759.25,A -85,B 0,C 180,E1 7883.761,E2 7883.761} C_VEL
LIN {X 0,Y 161.541,Z 773.479,A -85,B 0,C 180,E1 7878.492,E2 7878.492} C_VEL
LIN {X 0,Y 153.243,Z 785.875,A -85,B 0,C 180,E1 7872.493,E2 7872.493} C_VEL
LIN {X 0,Y 146.237,Z 796.866,A -85,B 0,C 180,E1 7865.527,E2 7865.527} C_VEL
LIN {X 0,Y 141.371,Z 805.456,A -85,B 0,C 180,E1 7858.28,E2 7858.28} C_VEL
LIN {X 0,Y 138.314,Z 812.644,A -85,B 0,C 180,E1 7850.299,E2 7850.299} C_VEL
LIN {X 0,Y 137.205,Z 817.761,A -85,B 0,C 180,E1 7842.624,E2 7842.624} C_VEL
LIN {X 0,Y 137.328,Z 821.025,A -85,B 0,C 180,E1 7835.427,E2 7835.427} C_VEL
LIN {X 0,Y 137.487,Z 822.518,A -85,B 0,C 180,E1 7829.996,E2 7829.996} C_VEL
LIN {X 0,Y 137.105,Z 823.122,A -85,B 0,C 180,E1 7824.556,E2 7824.556} C_VEL
LIN {X 0,Y 136.812,Z 822.793,A -85,B 0,C 180,E1 7817.331,E2 7817.331} C_VEL
LIN {X 0,Y 138.39,Z 820.912,A -85,B 0,C 180,E1 7807.929,E2 7807.929} C_VEL
LIN {X 0,Y 143.505,Z 817.031,A -85,B 0,C 180,E1 7798.023,E2 7798.023} C_VEL
LIN {X 0,Y 154.162,Z 810.719,A -85,B 0,C 180,E1 7787.579,E2 7787.579} C_VEL
LIN {X 0,Y 171.252,Z 801.908,A -85,B 0,C 180,E1 7777.978,E2 7777.978} C_VEL
LIN {X 0,Y 181.865,Z 796.736,A -85,B 0,C 180,E1 7773.88,E2 7773.88} C_VEL
LIN {X 0,Y 163.26,Z 800.839,A -85,B 0,C 180,E1 7765.39,E2 7765.39} C_VEL
LIN {X 0,Y 149.891,Z 802.957,A -85,B 0,C 180,E1 7755.48,E2 7755.48} C_VEL
LIN {X 0,Y 142.02,Z 803.157,A -85,B 0,C 180,E1 7745.257,E2 7745.257} C_VEL
LIN {X 0,Y 138.42,Z 801.755,A -85,B 0,C 180,E1 7735.863,E2 7735.863} C_VEL
LIN {X 0,Y 137.196,Z 799.328,A -85,B 0,C 180,E1 7727.377,E2 7727.377} C_VEL
LIN {X 0,Y 137.042,Z 796.276,A -85,B 0,C 180,E1 7720.262,E2 7720.262} C_VEL
LIN {X 0,Y 137.694,Z 792.06,A -85,B 0,C 180,E1 7712.783,E2 7712.783} C_VEL
LIN {X 0,Y 139.867,Z 785.791,A -85,B 0,C 180,E1 7704.588,E2 7704.588} C_VEL
LIN {X 0,Y 143.981,Z 777.786,A -85,B 0,C 180,E1 7696.577,E2 7696.577} C_VEL
LIN {X 0,Y 149.853,Z 768.339,A -85,B 0,C 180,E1 7689.297,E2 7689.297} C_VEL
LIN {X 0,Y 157.617,Z 756.69,A -85,B 0,C 180,E1 7682.478,E2 7682.478} C_VEL
LIN {X 0,Y 166.1,Z 744.137,A -85,B 0,C 180,E1 7676.842,E2 7676.842} C_VEL
LIN {X 0,Y 175.885,Z 729.341,A -85,B 0,C 180,E1 7671.688,E2 7671.688} C_VEL
LIN {X 0,Y 185.934,Z 713.32,A -85,B 0,C 180,E1 7667.368,E2 7667.368} C_VEL
LIN {X 0,Y 196.214,Z 695.659,A -85,B 0,C 180,E1 7663.657,E2 7663.657} C_VEL
LIN {X 0,Y 206.407,Z 676.323,A -85,B 0,C 180,E1 7660.497,E2 7660.497} C_VEL
LIN {X 0,Y 215.991,Z 655.847,A -85,B 0,C 180,E1 7657.881,E2 7657.881} C_VEL
LIN {X 0,Y 224.593,Z 634.937,A -85,B 0,C 180,E1 7655.784,E2 7655.784} C_VEL
LIN {X 0,Y 232.521,Z 612.541,A -85,B 0,C 180,E1 7654.025,E2 7654.025} C_VEL
LIN {X 0,Y 239.419,Z 589.145,A -85,B 0,C 180,E1 7652.604,E2 7652.604} C_VEL
LIN {X 0,Y 245.032,Z 565.444,A -85,B 0,C 180,E1 7651.519,E2 7651.519} C_VEL
LIN {X 0,Y 249.503,Z 540.604,A -85,B 0,C 180,E1 7650.7,E2 7650.7} C_VEL
LIN {X 0,Y 263.773,Z 448.667,A -85,B 0,C 180,E1 7648.21,E2 7648.21} C_VEL
LIN {X 0,Y 256.285,Z 436.455,A -85,B 0,C 180,E1 7643.956,E2 7643.956} C_VEL
LIN {X 0,Y 249.028,Z 425.015,A -85,B 0,C 180,E1 7639.184,E2 7639.184} C_VEL
LIN {X 0,Y 242.656,Z 415.61,A -85,B 0,C 180,E1 7634.29,E2 7634.29} C_VEL
LIN {X 0,Y 238.815,Z 410.129,A -85,B 0,C 180,E1 7630.815,E2 7630.815} C_VEL
LIN {X 0,Y 235.763,Z 405.785,A -85,B 0,C 180,E1 7627.738,E2 7627.738} C_VEL
LIN {X 0,Y 232.361,Z 401.018,A -85,B 0,C 180,E1 7623.694,E2 7623.694} C_VEL
LIN {X 0,Y 229.239,Z 396.458,A -85,B 0,C 180,E1 7619.111,E2 7619.111} C_VEL
LIN {X 0,Y 225.967,Z 392.462,A -85,B 0,C 180,E1 7612.786,E2 7612.786} C_VEL
LIN {X 0,Y 225.022,Z 390.387,A -85,B 0,C 180,E1 7609.834,E2 7609.834} C_VEL
LIN {X 0,Y 223.421,Z 389.371,A -85,B 0,C 180,E1 7603.163,E2 7603.163} C_VEL
LIN {X 0,Y 223.266,Z 389.281,A -85,B 0,C 180,E1 7596.551,E2 7596.551} C_VEL
LIN {X 0,Y 224.592,Z 390.191,A -85,B 0,C 180,E1 7589.766,E2 7589.766} C_VEL
LIN {X 0,Y 225.285,Z 390.836,A -85,B 0,C 180,E1 7587.771,E2 7587.771} C_VEL
LIN {X 0,Y 227.511,Z 394.886,A -85,B 0,C 180,E1 7581.991,E2 7581.991} C_VEL
LIN {X 0,Y 229.183,Z 396.539,A -85,B 0,C 180,E1 7579.227,E2 7579.227} C_VEL
LIN {X 0,Y 232.642,Z 401.317,A -85,B 0,C 180,E1 7574.177,E2 7574.177} C_VEL
LIN {X 0,Y 237.182,Z 407.82,A -85,B 0,C 180,E1 7568.848,E2 7568.848} C_VEL
LIN {X 0,Y 241.201,Z 413.515,A -85,B 0,C 180,E1 7564.991,E2 7564.991} C_VEL
LIN {X 0,Y 245.057,Z 419.114,A -85,B 0,C 180,E1 7561.679,E2 7561.679} C_VEL
LIN {X 0,Y 248.817,Z 425.187,A -85,B 0,C 180,E1 7558.731,E2 7558.731} C_VEL
LIN {X 0,Y 254.713,Z 435.351,A -85,B 0,C 180,E1 7554.591,E2 7554.591} C_VEL
LIN {X 0,Y 261.455,Z 447.571,A -85,B 0,C 180,E1 7550.421,E2 7550.421} C_VEL
LIN {X 0,Y 266.129,Z 456.756,A -85,B 0,C 180,E1 7547.769,E2 7547.769} C_VEL
LIN {X 0,Y 245.615,Z 585.974,A -85,B 0,C 180,E1 7544.221,E2 7544.221} C_VEL
LIN {X 0,Y 240.163,Z 610.187,A -85,B 0,C 180,E1 7543.288,E2 7543.288} C_VEL
LIN {X 0,Y 233.198,Z 633.635,A -85,B 0,C 180,E1 7542.137,E2 7542.137} C_VEL
LIN {X 0,Y 225.19,Z 656.142,A -85,B 0,C 180,E1 7540.64,E2 7540.64} C_VEL
LIN {X 0,Y 216.196,Z 677.904,A -85,B 0,C 180,E1 7538.723,E2 7538.723} C_VEL
LIN {X 0,Y 206,Z 699.442,A -85,B 0,C 180,E1 7536.24,E2 7536.24} C_VEL
LIN {X 0,Y 202.246,Z 706.801,A -85,B 0,C 180,E1 7535.226,E2 7535.226} C_VEL
LIN {X 0,Y 198.21,Z 713.028,A -85,B 0,C 180,E1 7534.47,E2 7534.47} C_VEL
LIN {X 0,Y 185.261,Z 727.702,A -85,B 0,C 180,E1 7533.048,E2 7533.048} C_VEL
LIN {X 0,Y 181.05,Z 733.317,A -85,B 0,C 180,E1 7532.087,E2 7532.087} C_VEL
LIN {X 0,Y 170.492,Z 749.72,A -85,B 0,C 180,E1 7528.027,E2 7528.027} C_VEL
LIN {X 0,Y 160.083,Z 764.983,A -85,B 0,C 180,E1 7523.073,E2 7523.073} C_VEL
LIN {X 0,Y 150.775,Z 778.261,A -85,B 0,C 180,E1 7517.393,E2 7517.393} C_VEL
LIN {X 0,Y 142.568,Z 790.112,A -85,B 0,C 180,E1 7510.704,E2 7510.704} C_VEL
LIN {X 0,Y 136.073,Z 800.148,A -85,B 0,C 180,E1 7503.097,E2 7503.097} C_VEL
LIN {X 0,Y 131.832,Z 808.083,A -85,B 0,C 180,E1 7495.128,E2 7495.128} C_VEL
LIN {X 0,Y 129.682,Z 814.198,A -85,B 0,C 180,E1 7487.032,E2 7487.032} C_VEL
LIN {X 0,Y 129.237,Z 818.304,A -85,B 0,C 180,E1 7479.346,E2 7479.346} C_VEL
LIN {X 0,Y 129.512,Z 820.611,A -85,B 0,C 180,E1 7473.093,E2 7473.093} C_VEL
LIN {X 0,Y 129.473,Z 821.676,A -85,B 0,C 180,E1 7468.225,E2 7468.225} C_VEL
LIN {X 0,Y 128.99,Z 822.13,A -85,B 0,C 180,E1 7462.424,E2 7462.424} C_VEL
LIN {X 0,Y 129.053,Z 821.624,A -85,B 0,C 180,E1 7454.262,E2 7454.262} C_VEL
LIN {X 0,Y 132.034,Z 819.302,A -85,B 0,C 180,E1 7443.458,E2 7443.458} C_VEL
LIN {X 0,Y 139.528,Z 815.012,A -85,B 0,C 180,E1 7432.703,E2 7432.703} C_VEL
LIN {X 0,Y 153.46,Z 808.207,A -85,B 0,C 180,E1 7422.028,E2 7422.028} C_VEL
LIN {X 0,Y 171.456,Z 800.232,A -85,B 0,C 180,E1 7413.747,E2 7413.747} C_VEL
LIN {X 0,Y 152.562,Z 803.365,A -85,B 0,C 180,E1 7404.391,E2 7404.391} C_VEL
LIN {X 0,Y 139.731,Z 804.45,A -85,B 0,C 180,E1 7393.664,E2 7393.664} C_VEL
LIN {X 0,Y 132.801,Z 803.683,A -85,B 0,C 180,E1 7383.027,E2 7383.027} C_VEL
LIN {X 0,Y 129.88,Z 801.602,A -85,B 0,C 180,E1 7373.289,E2 7373.289} C_VEL
LIN {X 0,Y 129.102,Z 798.894,A -85,B 0,C 180,E1 7365.199,E2 7365.199} C_VEL
LIN {X 0,Y 129.197,Z 795.049,A -85,B 0,C 180,E1 7357.074,E2 7357.074} C_VEL
LIN {X 0,Y 130.415,Z 790.086,A -85,B 0,C 180,E1 7349.099,E2 7349.099} C_VEL
LIN {X 0,Y 133.545,Z 783.002,A -85,B 0,C 180,E1 7340.464,E2 7340.464} C_VEL
LIN {X 0,Y 138.517,Z 774.597,A -85,B 0,C 180,E1 7332.595,E2 7332.595} C_VEL
LIN {X 0,Y 145.534,Z 764.162,A -85,B 0,C 180,E1 7325.169,E2 7325.169} C_VEL
LIN {X 0,Y 153.902,Z 752.258,A -85,B 0,C 180,E1 7318.723,E2 7318.723} C_VEL
LIN {X 0,Y 163.841,Z 738.077,A -85,B 0,C 180,E1 7312.87,E2 7312.87} C_VEL
LIN {X 0,Y 174.071,Z 722.87,A -85,B 0,C 180,E1 7308.073,E2 7308.073} C_VEL
LIN {X 0,Y 184.475,Z 706.383,A -85,B 0,C 180,E1 7304.05,E2 7304.05} C_VEL
LIN {X 0,Y 195.235,Z 687.61,A -85,B 0,C 180,E1 7300.518,E2 7300.518} C_VEL
LIN {X 0,Y 205.359,Z 667.915,A -85,B 0,C 180,E1 7297.649,E2 7297.649} C_VEL
LIN {X 0,Y 214.516,Z 647.831,A -85,B 0,C 180,E1 7295.351,E2 7295.351} C_VEL
LIN {X 0,Y 223.421,Z 625.361,A -85,B 0,C 180,E1 7293.338,E2 7293.338} C_VEL
LIN {X 0,Y 231.144,Z 602.253,A -85,B 0,C 180,E1 7291.738,E2 7291.738} C_VEL
LIN {X 0,Y 237.584,Z 578.781,A -85,B 0,C 180,E1 7290.499,E2 7290.499} C_VEL
LIN {X 0,Y 242.705,Z 555.129,A -85,B 0,C 180,E1 7289.573,E2 7289.573} C_VEL
LIN {X 0,Y 259.146,Z 453.002,A -85,B 0,C 180,E1 7286.795,E2 7286.795} C_VEL
LIN {X 0,Y 251.557,Z 440.479,A -85,B 0,C 180,E1 7282.236,E2 7282.236} C_VEL
LIN {X 0,Y 245.277,Z 430.694,A -85,B 0,C 180,E1 7277.884,E2 7277.884} C_VEL
LIN {X 0,Y 239.984,Z 422.648,A -85,B 0,C 180,E1 7273.607,E2 7273.607} C_VEL
LIN {X 0,Y 236.386,Z 417.373,A -85,B 0,C 180,E1 7270.225,E2 7270.225} C_VEL
LIN {X 0,Y 233.482,Z 413.153,A -85,B 0,C 180,E1 7267.187,E2 7267.187} C_VEL
LIN {X 0,Y 230.35,Z 408.665,A -85,B 0,C 180,E1 7263.391,E2 7263.391} C_VEL
LIN {X 0,Y 227.262,Z 404.071,A -85,B 0,C 180,E1 7258.728,E2 7258.728} C_VEL
LIN {X 0,Y 224.001,Z 399.776,A -85,B 0,C 180,E1 7251.981,E2 7251.981} C_VEL
LIN {X 0,Y 223.208,Z 398.157,A -85,B 0,C 180,E1 7249.591,E2 7249.591} C_VEL
LIN {X 0,Y 221.656,Z 397.144,A -85,B 0,C 180,E1 7242.575,E2 7242.575} C_VEL
LIN {X 0,Y 221.577,Z 397.127,A -85,B 0,C 180,E1 7235.912,E2 7235.912} C_VEL
LIN {X 0,Y 223.158,Z 398.152,A -85,B 0,C 180,E1 7228.935,E2 7228.935} C_VEL
LIN {X 0,Y 223.826,Z 399.748,A -85,B 0,C 180,E1 7226.528,E2 7226.528} C_VEL
LIN {X 0,Y 226.339,Z 403.28,A -85,B 0,C 180,E1 7220.962,E2 7220.962} C_VEL
LIN {X 0,Y 227.296,Z 404.394,A -85,B 0,C 180,E1 7219.393,E2 7219.393} C_VEL
LIN {X 0,Y 231.256,Z 409.984,A -85,B 0,C 180,E1 7213.625,E2 7213.625} C_VEL
LIN {X 0,Y 235.097,Z 415.482,A -85,B 0,C 180,E1 7209.174,E2 7209.174} C_VEL
LIN {X 0,Y 238.833,Z 420.904,A -85,B 0,C 180,E1 7205.462,E2 7205.462} C_VEL
LIN {X 0,Y 242.575,Z 426.415,A -85,B 0,C 180,E1 7202.182,E2 7202.182} C_VEL
LIN {X 0,Y 246.207,Z 432.351,A -85,B 0,C 180,E1 7199.299,E2 7199.299} C_VEL
LIN {X 0,Y 252.024,Z 442.632,A -85,B 0,C 180,E1 7195.104,E2 7195.104} C_VEL
LIN {X 0,Y 258.499,Z 454.624,A -85,B 0,C 180,E1 7190.985,E2 7190.985} C_VEL
LIN {X 0,Y 261.544,Z 460.769,A -85,B 0,C 180,E1 7189.18,E2 7189.18} C_VEL
LIN {X 0,Y 241.045,Z 586.036,A -85,B 0,C 180,E1 7185.767,E2 7185.767} C_VEL
LIN {X 0,Y 235.399,Z 610.387,A -85,B 0,C 180,E1 7184.838,E2 7184.838} C_VEL
LIN {X 0,Y 228.146,Z 634.106,A -85,B 0,C 180,E1 7183.682,E2 7183.682} C_VEL
LIN {X 0,Y 220.138,Z 655.975,A -85,B 0,C 180,E1 7182.236,E2 7182.236} C_VEL
LIN {X 0,Y 211.2,Z 677.066,A -85,B 0,C 180,E1 7180.397,E2 7180.397} C_VEL
LIN {X 0,Y 201.042,Z 698.041,A -85,B 0,C 180,E1 7178.012,E2 7178.012} C_VEL
LIN {X 0,Y 190.599,Z 717.25,A -85,B 0,C 180,E1 7175.158,E2 7175.158} C_VEL
LIN {X 0,Y 181.05,Z 733.317,A -85,B 0,C 180,E1 7172.087,E2 7172.087} C_VEL
LIN {X 0,Y 176.783,Z 738.917,A -85,B 0,C 180,E1 7171.037,E2 7171.037} C_VEL
LIN {X 0,Y 162.356,Z 752.708,A -85,B 0,C 180,E1 7168.521,E2 7168.521} C_VEL
LIN {X 0,Y 158.672,Z 756.995,A -85,B 0,C 180,E1 7167.282,E2 7167.282} C_VEL
LIN {X 0,Y 147.977,Z 771.764,A -85,B 0,C 180,E1 7161.602,E2 7161.602} C_VEL
LIN {X 0,Y 139.08,Z 783.91,A -85,B 0,C 180,E1 7155.368,E2 7155.368} C_VEL
LIN {X 0,Y 131.478,Z 794.641,A -85,B 0,C 180,E1 7148.017,E2 7148.017} C_VEL
LIN {X 0,Y 125.97,Z 803.346,A -85,B 0,C 180,E1 7139.998,E2 7139.998} C_VEL
LIN {X 0,Y 122.519,Z 810.643,A -85,B 0,C 180,E1 7131.038,E2 7131.038} C_VEL
LIN {X 0,Y 121.353,Z 815.527,A -85,B 0,C 180,E1 7122.849,E2 7122.849} C_VEL
LIN {X 0,Y 121.488,Z 818.838,A -85,B 0,C 180,E1 7115.173,E2 7115.173} C_VEL
LIN {X 0,Y 121.625,Z 820.332,A -85,B 0,C 180,E1 7109.524,E2 7109.524} C_VEL
LIN {X 0,Y 121.13,Z 821.05,A -85,B 0,C 180,E1 7103.359,E2 7103.359} C_VEL
LIN {X 0,Y 121.145,Z 820.781,A -85,B 0,C 180,E1 7093.698,E2 7093.698} C_VEL
LIN {X 0,Y 123.816,Z 819.073,A -85,B 0,C 180,E1 7083.627,E2 7083.627} C_VEL
LIN {X 0,Y 132.372,Z 814.937,A -85,B 0,C 180,E1 7071.171,E2 7071.171} C_VEL
LIN {X 0,Y 147.462,Z 808.62,A -85,B 0,C 180,E1 7059.982,E2 7059.982} C_VEL
LIN {X 0,Y 160.904,Z 803.24,A -85,B 0,C 180,E1 7053.581,E2 7053.581} C_VEL
LIN {X 0,Y 142.839,Z 805.278,A -85,B 0,C 180,E1 7043.959,E2 7043.959} C_VEL
LIN {X 0,Y 130.945,Z 805.487,A -85,B 0,C 180,E1 7033.248,E2 7033.248} C_VEL
LIN {X 0,Y 124.199,Z 804.057,A -85,B 0,C 180,E1 7021.851,E2 7021.851} C_VEL
LIN {X 0,Y 121.668,Z 801.656,A -85,B 0,C 180,E1 7011.976,E2 7011.976} C_VEL
LIN {X 0,Y 121.053,Z 798.433,A -85,B 0,C 180,E1 7003.374,E2 7003.374} C_VEL
LIN {X 0,Y 121.314,Z 794.686,A -85,B 0,C 180,E1 6995.671,E2 6995.671} C_VEL
LIN {X 0,Y 123.069,Z 788.836,A -85,B 0,C 180,E1 6986.473,E2 6986.473} C_VEL
LIN {X 0,Y 126.974,Z 781.239,A -85,B 0,C 180,E1 6977.384,E2 6977.384} C_VEL
LIN {X 0,Y 132.868,Z 772.099,A -85,B 0,C 180,E1 6969.197,E2 6969.197} C_VEL
LIN {X 0,Y 140.884,Z 760.928,A -85,B 0,C 180,E1 6961.622,E2 6961.622} C_VEL
LIN {X 0,Y 150.215,Z 748.284,A -85,B 0,C 180,E1 6955.159,E2 6955.159} C_VEL
LIN {X 0,Y 160.483,Z 734.078,A -85,B 0,C 180,E1 6949.663,E2 6949.663} C_VEL
LIN {X 0,Y 171.726,Z 717.56,A -85,B 0,C 180,E1 6944.847,E2 6944.847} C_VEL
LIN {X 0,Y 182.368,Z 700.58,A -85,B 0,C 180,E1 6941.066,E2 6941.066} C_VEL
LIN {X 0,Y 193.06,Z 681.861,A -85,B 0,C 180,E1 6937.837,E2 6937.837} C_VEL
LIN {X 0,Y 203.739,Z 660.865,A -85,B 0,C 180,E1 6935.035,E2 6935.035} C_VEL
LIN {X 0,Y 213.474,Z 638.932,A -85,B 0,C 180,E1 6932.775,E2 6932.775} C_VEL
LIN {X 0,Y 221.798,Z 617.153,A -85,B 0,C 180,E1 6931.036,E2 6931.036} C_VEL
LIN {X 0,Y 228.953,Z 594.964,A -85,B 0,C 180,E1 6929.654,E2 6929.654} C_VEL
LIN {X 0,Y 235.423,Z 570.038,A -85,B 0,C 180,E1 6928.484,E2 6928.484} C_VEL
LIN {X 0,Y 240.403,Z 544.645,A -85,B 0,C 180,E1 6927.634,E2 6927.634} C_VEL
LIN {X 0,Y 254.656,Z 457.429,A -85,B 0,C 180,E1 6925.329,E2 6925.329} C_VEL
LIN {X 0,Y 248.011,Z 446.358,A -85,B 0,C 180,E1 6921.138,E2 6921.138} C_VEL
LIN {X 0,Y 242.283,Z 437.248,A -85,B 0,C 180,E1 6917.005,E2 6917.005} C_VEL
LIN {X 0,Y 237.295,Z 429.592,A -85,B 0,C 180,E1 6912.848,E2 6912.848} C_VEL
LIN {X 0,Y 234.068,Z 424.788,A -85,B 0,C 180,E1 6909.76,E2 6909.76} C_VEL
LIN {X 0,Y 231.288,Z 420.603,A -85,B 0,C 180,E1 6906.702,E2 6906.702} C_VEL
LIN {X 0,Y 228.144,Z 416.101,A -85,B 0,C 180,E1 6902.821,E2 6902.821} C_VEL
LIN {X 0,Y 224.873,Z 411.215,A -85,B 0,C 180,E1 6897.642,E2 6897.642} C_VEL
LIN {X 0,Y 222.043,Z 407.273,A -85,B 0,C 180,E1 6891.436,E2 6891.436} C_VEL
LIN {X 0,Y 221.397,Z 405.928,A -85,B 0,C 180,E1 6889.344,E2 6889.344} C_VEL
LIN {X 0,Y 219.847,Z 404.915,A -85,B 0,C 180,E1 6881.949,E2 6881.949} C_VEL
LIN {X 0,Y 219.881,Z 404.976,A -85,B 0,C 180,E1 6875.521,E2 6875.521} C_VEL
LIN {X 0,Y 221.553,Z 406.076,A -85,B 0,C 180,E1 6868.574,E2 6868.574} C_VEL
LIN {X 0,Y 223.725,Z 410.259,A -85,B 0,C 180,E1 6862.599,E2 6862.599} C_VEL
LIN {X 0,Y 225.272,Z 411.972,A -85,B 0,C 180,E1 6859.798,E2 6859.798} C_VEL
LIN {X 0,Y 229.182,Z 417.574,A -85,B 0,C 180,E1 6854.009,E2 6854.009} C_VEL
LIN {X 0,Y 232.902,Z 423.032,A -85,B 0,C 180,E1 6849.566,E2 6849.566} C_VEL
LIN {X 0,Y 236.656,Z 428.589,A -85,B 0,C 180,E1 6845.755,E2 6845.755} C_VEL
LIN {X 0,Y 240.328,Z 434.036,A -85,B 0,C 180,E1 6842.512,E2 6842.512} C_VEL
LIN {X 0,Y 244.702,Z 441.42,A -85,B 0,C 180,E1 6839.002,E2 6839.002} C_VEL
LIN {X 0,Y 250.998,Z 453.002,A -85,B 0,C 180,E1 6834.471,E2 6834.471} C_VEL
LIN {X 0,Y 257.053,Z 464.644,A -85,B 0,C 180,E1 6830.637,E2 6830.637} C_VEL
LIN {X 0,Y 236.815,Z 585.11,A -85,B 0,C 180,E1 6827.399,E2 6827.399} C_VEL
LIN {X 0,Y 231.034,Z 609.458,A -85,B 0,C 180,E1 6826.482,E2 6826.482} C_VEL
LIN {X 0,Y 223.714,Z 632.907,A -85,B 0,C 180,E1 6825.366,E2 6825.366} C_VEL
LIN {X 0,Y 215.38,Z 655.185,A -85,B 0,C 180,E1 6823.924,E2 6823.924} C_VEL
LIN {X 0,Y 205.974,Z 676.808,A -85,B 0,C 180,E1 6822.06,E2 6822.06} C_VEL
LIN {X 0,Y 195.256,Z 698.275,A -85,B 0,C 180,E1 6819.618,E2 6819.618} C_VEL
LIN {X 0,Y 184.069,Z 718.137,A -85,B 0,C 180,E1 6816.627,E2 6816.627} C_VEL
LIN {X 0,Y 173.141,Z 735.773,A -85,B 0,C 180,E1 6813.119,E2 6813.119} C_VEL
LIN {X 0,Y 161.943,Z 752.415,A -85,B 0,C 180,E1 6808.755,E2 6808.755} C_VEL
LIN {X 0,Y 158.672,Z 756.995,A -85,B 0,C 180,E1 6807.282,E2 6807.282} C_VEL
LIN {X 0,Y 154.32,Z 761.937,A -85,B 0,C 180,E1 6805.764,E2 6805.764} C_VEL
LIN {X 0,Y 139.818,Z 773.824,A -85,B 0,C 180,E1 6801.85,E2 6801.85} C_VEL
LIN {X 0,Y 136.248,Z 777.467,A -85,B 0,C 180,E1 6800.072,E2 6800.072} C_VEL
LIN {X 0,Y 127.547,Z 788.896,A -85,B 0,C 180,E1 6792.994,E2 6792.994} C_VEL
LIN {X 0,Y 120.655,Z 798.525,A -85,B 0,C 180,E1 6784.866,E2 6784.866} C_VEL
LIN {X 0,Y 115.87,Z 806.693,A -85,B 0,C 180,E1 6775.554,E2 6775.554} C_VEL
LIN {X 0,Y 113.694,Z 812.709,A -85,B 0,C 180,E1 6766.339,E2 6766.339} C_VEL
LIN {X 0,Y 113.446,Z 816.682,A -85,B 0,C 180,E1 6757.592,E2 6757.592} C_VEL
LIN {X 0,Y 113.735,Z 818.605,A -85,B 0,C 180,E1 6751.506,E2 6751.506} C_VEL
LIN {X 0,Y 113.456,Z 819.633,A -85,B 0,C 180,E1 6745.952,E2 6745.952} C_VEL
LIN {X 0,Y 112.975,Z 820.019,A -85,B 0,C 180,E1 6737.212,E2 6737.212} C_VEL
LIN {X 0,Y 114.707,Z 819.13,A -85,B 0,C 180,E1 6726.356,E2 6726.356} C_VEL
LIN {X 0,Y 121.91,Z 816.1,A -85,B 0,C 180,E1 6713.217,E2 6713.217} C_VEL
LIN {X 0,Y 135.683,Z 811.04,A -85,B 0,C 180,E1 6701.261,E2 6701.261} C_VEL
LIN {X 0,Y 150.469,Z 805.765,A -85,B 0,C 180,E1 6693.477,E2 6693.477} C_VEL
LIN {X 0,Y 132.573,Z 806.837,A -85,B 0,C 180,E1 6683.096,E2 6683.096} C_VEL
LIN {X 0,Y 121.152,Z 806.152,A -85,B 0,C 180,E1 6671.43,E2 6671.43} C_VEL
LIN {X 0,Y 115.303,Z 803.994,A -85,B 0,C 180,E1 6659.51,E2 6659.51} C_VEL
LIN {X 0,Y 113.404,Z 801.175,A -85,B 0,C 180,E1 6649.851,E2 6649.851} C_VEL
LIN {X 0,Y 113.047,Z 797.794,A -85,B 0,C 180,E1 6641.165,E2 6641.165} C_VEL
LIN {X 0,Y 113.822,Z 792.816,A -85,B 0,C 180,E1 6631.691,E2 6631.691} C_VEL
LIN {X 0,Y 116.583,Z 786.168,A -85,B 0,C 180,E1 6621.876,E2 6621.876} C_VEL
LIN {X 0,Y 121.471,Z 778.04,A -85,B 0,C 180,E1 6612.908,E2 6612.908} C_VEL
LIN {X 0,Y 128.657,Z 768.012,A -85,B 0,C 180,E1 6604.548,E2 6604.548} C_VEL
LIN {X 0,Y 137.99,Z 755.823,A -85,B 0,C 180,E1 6596.986,E2 6596.986} C_VEL
LIN {X 0,Y 147.894,Z 742.943,A -85,B 0,C 180,E1 6591.001,E2 6591.001} C_VEL
LIN {X 0,Y 159.133,Z 727.594,A -85,B 0,C 180,E1 6585.678,E2 6585.678} C_VEL
LIN {X 0,Y 170.311,Z 711.152,A -85,B 0,C 180,E1 6581.387,E2 6581.387} C_VEL
LIN {X 0,Y 181.624,Z 692.991,A -85,B 0,C 180,E1 6577.77,E2 6577.77} C_VEL
LIN {X 0,Y 192.619,Z 673.314,A -85,B 0,C 180,E1 6574.759,E2 6574.759} C_VEL
LIN {X 0,Y 202.657,Z 653.031,A -85,B 0,C 180,E1 6572.355,E2 6572.355} C_VEL
LIN {X 0,Y 211.956,Z 631.484,A -85,B 0,C 180,E1 6570.369,E2 6570.369} C_VEL
LIN {X 0,Y 220.505,Z 608.065,A -85,B 0,C 180,E1 6568.703,E2 6568.703} C_VEL
LIN {X 0,Y 227.63,Z 584.24,A -85,B 0,C 180,E1 6567.415,E2 6567.415} C_VEL
LIN {X 0,Y 233.431,Z 559.695,A -85,B 0,C 180,E1 6566.439,E2 6566.439} C_VEL
LIN {X 0,Y 242.017,Z 510.591,A -85,B 0,C 180,E1 6565.091,E2 6565.091} C_VEL
LIN {X 0,Y 250.241,Z 461.775,A -85,B 0,C 180,E1 6563.809,E2 6563.809} C_VEL
LIN {X 0,Y 243.055,Z 449.76,A -85,B 0,C 180,E1 6558.975,E2 6558.975} C_VEL
LIN {X 0,Y 237.272,Z 440.593,A -85,B 0,C 180,E1 6554.426,E2 6554.426} C_VEL
LIN {X 0,Y 232.377,Z 432.987,A -85,B 0,C 180,E1 6549.869,E2 6549.869} C_VEL
LIN {X 0,Y 228.906,Z 427.844,A -85,B 0,C 180,E1 6546.035,E2 6546.035} C_VEL
LIN {X 0,Y 226.023,Z 423.601,A -85,B 0,C 180,E1 6542.326,E2 6542.326} C_VEL
LIN {X 0,Y 223.006,Z 418.956,A -85,B 0,C 180,E1 6537.44,E2 6537.44} C_VEL
LIN {X 0,Y 220.168,Z 415.012,A -85,B 0,C 180,E1 6531.196,E2 6531.196} C_VEL
LIN {X 0,Y 219.531,Z 413.681,A -85,B 0,C 180,E1 6529.02,E2 6529.02} C_VEL
LIN {X 0,Y 218.016,Z 412.688,A -85,B 0,C 180,E1 6521.325,E2 6521.325} C_VEL
LIN {X 0,Y 218.165,Z 412.81,A -85,B 0,C 180,E1 6515.267,E2 6515.267} C_VEL
LIN {X 0,Y 219.746,Z 413.955,A -85,B 0,C 180,E1 6508.668,E2 6508.668} C_VEL
LIN {X 0,Y 222.013,Z 418.168,A -85,B 0,C 180,E1 6502.503,E2 6502.503} C_VEL
LIN {X 0,Y 223.267,Z 419.593,A -85,B 0,C 180,E1 6500.167,E2 6500.167} C_VEL
LIN {X 0,Y 227.064,Z 425.173,A -85,B 0,C 180,E1 6494.374,E2 6494.374} C_VEL
LIN {X 0,Y 230.605,Z 430.443,A -85,B 0,C 180,E1 6490.051,E2 6490.051} C_VEL
LIN {X 0,Y 234.242,Z 435.895,A -85,B 0,C 180,E1 6486.288,E2 6486.288} C_VEL
LIN {X 0,Y 238.334,Z 442.009,A -85,B 0,C 180,E1 6482.642,E2 6482.642} C_VEL
LIN {X 0,Y 244.013,Z 452.216,A -85,B 0,C 180,E1 6478.048,E2 6478.048} C_VEL
LIN {X 0,Y 250.779,Z 465.101,A -85,B 0,C 180,E1 6473.3,E2 6473.3} C_VEL
LIN {X 0,Y 252.574,Z 468.985,A -85,B 0,C 180,E1 6472.116,E2 6472.116} C_VEL
LIN {X 0,Y 232.478,Z 584.941,A -85,B 0,C 180,E1 6469.04,E2 6469.04} C_VEL
LIN {X 0,Y 226.542,Z 609.325,A -85,B 0,C 180,E1 6468.14,E2 6468.14} C_VEL
LIN {X 0,Y 219.032,Z 632.812,A -85,B 0,C 180,E1 6467.045,E2 6467.045} C_VEL
LIN {X 0,Y 210.539,Z 654.966,A -85,B 0,C 180,E1 6465.637,E2 6465.637} C_VEL
LIN {X 0,Y 200.931,Z 676.506,A -85,B 0,C 180,E1 6463.807,E2 6463.807} C_VEL
LIN {X 0,Y 190.315,Z 697.257,A -85,B 0,C 180,E1 6461.483,E2 6461.483} C_VEL
LIN {X 0,Y 179.266,Z 716.439,A -85,B 0,C 180,E1 6458.651,E2 6458.651} C_VEL
LIN {X 0,Y 168.355,Z 733.635,A -85,B 0,C 180,E1 6455.311,E2 6455.311} C_VEL
LIN {X 0,Y 156.673,Z 750.423,A -85,B 0,C 180,E1 6450.954,E2 6450.954} C_VEL
LIN {X 0,Y 145.994,Z 764.773,A -85,B 0,C 180,E1 6445.956,E2 6445.956} C_VEL
LIN {X 0,Y 136.248,Z 777.467,A -85,B 0,C 180,E1 6440.072,E2 6440.072} C_VEL
LIN {X 0,Y 132.107,Z 781.641,A -85,B 0,C 180,E1 6437.884,E2 6437.884} C_VEL
LIN {X 0,Y 118.511,Z 791.304,A -85,B 0,C 180,E1 6431.853,E2 6431.853} C_VEL
LIN {X 0,Y 115.506,Z 794.232,A -85,B 0,C 180,E1 6429.308,E2 6429.308} C_VEL
LIN {X 0,Y 109.667,Z 802.758,A -85,B 0,C 180,E1 6420.089,E2 6420.089} C_VEL
LIN {X 0,Y 106.288,Z 809.727,A -85,B 0,C 180,E1 6409.789,E2 6409.789} C_VEL
LIN {X 0,Y 105.462,Z 814.386,A -85,B 0,C 180,E1 6400.372,E2 6400.372} C_VEL
LIN {X 0,Y 105.785,Z 817.069,A -85,B 0,C 180,E1 6392.703,E2 6392.703} C_VEL
LIN {X 0,Y 105.672,Z 818.166,A -85,B 0,C 180,E1 6387.283,E2 6387.283} C_VEL
LIN {X 0,Y 105.052,Z 818.901,A -85,B 0,C 180,E1 6379.021,E2 6379.021} C_VEL
LIN {X 0,Y 106.687,Z 818.418,A -85,B 0,C 180,E1 6366.229,E2 6366.229} C_VEL
LIN {X 0,Y 113.079,Z 816.262,A -85,B 0,C 180,E1 6353.584,E2 6353.584} C_VEL
LIN {X 0,Y 127.964,Z 811.559,A -85,B 0,C 180,E1 6340.022,E2 6340.022} C_VEL
LIN {X 0,Y 139.989,Z 807.846,A -85,B 0,C 180,E1 6333.37,E2 6333.37} C_VEL
LIN {X 0,Y 122.301,Z 807.964,A -85,B 0,C 180,E1 6322.097,E2 6322.097} C_VEL
LIN {X 0,Y 111.142,Z 806.297,A -85,B 0,C 180,E1 6308.804,E2 6308.804} C_VEL
LIN {X 0,Y 106.503,Z 803.572,A -85,B 0,C 180,E1 6296.778,E2 6296.778} C_VEL
LIN {X 0,Y 105.183,Z 800.262,A -85,B 0,C 180,E1 6286.82,E2 6286.82} C_VEL
LIN {X 0,Y 105.129,Z 796.627,A -85,B 0,C 180,E1 6278.236,E2 6278.236} C_VEL
LIN {X 0,Y 106.465,Z 791.291,A -85,B 0,C 180,E1 6268.279,E2 6268.279} C_VEL
LIN {X 0,Y 110.049,Z 784.103,A -85,B 0,C 180,E1 6258.168,E2 6258.168} C_VEL
LIN {X 0,Y 116.272,Z 774.993,A -85,B 0,C 180,E1 6248.519,E2 6248.519} C_VEL
LIN {X 0,Y 124.222,Z 764.831,A -85,B 0,C 180,E1 6240.475,E2 6240.475} C_VEL
LIN {X 0,Y 134.156,Z 752.452,A -85,B 0,C 180,E1 6233.271,E2 6233.271} C_VEL
LIN {X 0,Y 144.665,Z 739.067,A -85,B 0,C 180,E1 6227.508,E2 6227.508} C_VEL
LIN {X 0,Y 156.59,Z 723.052,A -85,B 0,C 180,E1 6222.359,E2 6222.359} C_VEL
LIN {X 0,Y 168.544,Z 705.643,A -85,B 0,C 180,E1 6218.189,E2 6218.189} C_VEL
LIN {X 0,Y 179.623,Z 687.866,A -85,B 0,C 180,E1 6214.938,E2 6214.938} C_VEL
LIN {X 0,Y 191.078,Z 667.222,A -85,B 0,C 180,E1 6212.054,E2 6212.054} C_VEL
LIN {X 0,Y 201.682,Z 645.288,A -85,B 0,C 180,E1 6209.719,E2 6209.719} C_VEL
LIN {X 0,Y 211.098,Z 622.516,A -85,B 0,C 180,E1 6207.862,E2 6207.862} C_VEL
LIN {X 0,Y 218.719,Z 600.542,A -85,B 0,C 180,E1 6206.487,E2 6206.487} C_VEL
LIN {X 0,Y 225.512,Z 576.675,A -85,B 0,C 180,E1 6205.351,E2 6205.351} C_VEL
LIN {X 0,Y 230.964,Z 552.032,A -85,B 0,C 180,E1 6204.497,E2 6204.497} C_VEL
LIN {X 0,Y 245.908,Z 466.363,A -85,B 0,C 180,E1 6202.291,E2 6202.291} C_VEL
LIN {X 0,Y 239.88,Z 456.129,A -85,B 0,C 180,E1 6198.035,E2 6198.035} C_VEL
LIN {X 0,Y 234.375,Z 447.235,A -85,B 0,C 180,E1 6193.535,E2 6193.535} C_VEL
LIN {X 0,Y 229.771,Z 440.015,A -85,B 0,C 180,E1 6189.098,E2 6189.098} C_VEL
LIN {X 0,Y 226.767,Z 435.417,A -85,B 0,C 180,E1 6185.67,E2 6185.67} C_VEL
LIN {X 0,Y 223.97,Z 431.167,A -85,B 0,C 180,E1 6181.906,E2 6181.906} C_VEL
LIN {X 0,Y 221.087,Z 426.652,A -85,B 0,C 180,E1 6177.136,E2 6177.136} C_VEL
LIN {X 0,Y 218.201,Z 422.493,A -85,B 0,C 180,E1 6170.627,E2 6170.627} C_VEL
LIN {X 0,Y 217.721,Z 421.461,A -85,B 0,C 180,E1 6168.857,E2 6168.857} C_VEL
LIN {X 0,Y 216.258,Z 420.494,A -85,B 0,C 180,E1 6161.382,E2 6161.382} C_VEL
LIN {X 0,Y 216.414,Z 420.629,A -85,B 0,C 180,E1 6155.144,E2 6155.144} C_VEL
LIN {X 0,Y 217.911,Z 421.793,A -85,B 0,C 180,E1 6148.797,E2 6148.797} C_VEL
LIN {X 0,Y 220.145,Z 425.909,A -85,B 0,C 180,E1 6142.705,E2 6142.705} C_VEL
LIN {X 0,Y 221.287,Z 427.266,A -85,B 0,C 180,E1 6140.494,E2 6140.494} C_VEL
LIN {X 0,Y 224.912,Z 432.694,A -85,B 0,C 180,E1 6134.806,E2 6134.806} C_VEL
LIN {X 0,Y 228.395,Z 437.972,A -85,B 0,C 180,E1 6130.464,E2 6130.464} C_VEL
LIN {X 0,Y 232,Z 443.443,A -85,B 0,C 180,E1 6126.679,E2 6126.679} C_VEL
LIN {X 0,Y 236,Z 449.588,A -85,B 0,C 180,E1 6123.032,E2 6123.032} C_VEL
LIN {X 0,Y 241.443,Z 459.662,A -85,B 0,C 180,E1 6118.514,E2 6118.514} C_VEL
LIN {X 0,Y 247.9,Z 472.284,A -85,B 0,C 180,E1 6113.861,E2 6113.861} C_VEL
LIN {X 0,Y 248.166,Z 473.191,A -85,B 0,C 180,E1 6113.643,E2 6113.643} C_VEL
LIN {X 0,Y 228.422,Z 584.384,A -85,B 0,C 180,E1 6110.756,E2 6110.756} C_VEL
LIN {X 0,Y 222.413,Z 608.583,A -85,B 0,C 180,E1 6109.884,E2 6109.884} C_VEL
LIN {X 0,Y 214.777,Z 631.948,A -85,B 0,C 180,E1 6108.828,E2 6108.828} C_VEL
LIN {X 0,Y 206.348,Z 653.488,A -85,B 0,C 180,E1 6107.503,E2 6107.503} C_VEL
LIN {X 0,Y 196.528,Z 675.087,A -85,B 0,C 180,E1 6105.726,E2 6105.726} C_VEL
LIN {X 0,Y 185.317,Z 696.49,A -85,B 0,C 180,E1 6103.38,E2 6103.38} C_VEL
LIN {X 0,Y 173.877,Z 715.789,A -85,B 0,C 180,E1 6100.56,E2 6100.56} C_VEL
LIN {X 0,Y 162.477,Z 733.181,A -85,B 0,C 180,E1 6097.184,E2 6097.184} C_VEL
LIN {X 0,Y 150.547,Z 749.749,A -85,B 0,C 180,E1 6092.859,E2 6092.859} C_VEL
LIN {X 0,Y 139.444,Z 764.099,A -85,B 0,C 180,E1 6087.781,E2 6087.781} C_VEL
LIN {X 0,Y 128.971,Z 777.142,A -85,B 0,C 180,E1 6081.529,E2 6081.529} C_VEL
LIN {X 0,Y 119.672,Z 788.771,A -85,B 0,C 180,E1 6073.897,E2 6073.897} C_VEL
LIN {X 0,Y 115.506,Z 794.232,A -85,B 0,C 180,E1 6069.308,E2 6069.308} C_VEL
LIN {X 0,Y 112.131,Z 797.436,A -85,B 0,C 180,E1 6066.17,E2 6066.17} C_VEL
LIN {X 0,Y 104.169,Z 802.4,A -85,B 0,C 180,E1 6060.251,E2 6060.251} C_VEL
LIN {X 0,Y 99.925,Z 805.553,A -85,B 0,C 180,E1 6055.441,E2 6055.441} C_VEL
LIN {X 0,Y 99.199,Z 806.634,A -85,B 0,C 180,E1 6053.672,E2 6053.672} C_VEL
LIN {X 0,Y 97.602,Z 812.036,A -85,B 0,C 180,E1 6043.019,E2 6043.019} C_VEL
LIN {X 0,Y 97.794,Z 815.087,A -85,B 0,C 180,E1 6034.686,E2 6034.686} C_VEL
LIN {X 0,Y 97.897,Z 816.57,A -85,B 0,C 180,E1 6028.824,E2 6028.824} C_VEL
LIN {X 0,Y 97.221,Z 817.558,A -85,B 0,C 180,E1 6020.902,E2 6020.902} C_VEL
LIN {X 0,Y 97.967,Z 817.7,A -85,B 0,C 180,E1 6009.065,E2 6009.065} C_VEL
LIN {X 0,Y 103.809,Z 816.301,A -85,B 0,C 180,E1 5994.691,E2 5994.691} C_VEL
LIN {X 0,Y 117.358,Z 812.703,A -85,B 0,C 180,E1 5980.683,E2 5980.683} C_VEL
LIN {X 0,Y 129.477,Z 809.481,A -85,B 0,C 180,E1 5973.255,E2 5973.255} C_VEL
LIN {X 0,Y 112.023,Z 808.658,A -85,B 0,C 180,E1 5960.924,E2 5960.924} C_VEL
LIN {X 0,Y 102.075,Z 806.328,A -85,B 0,C 180,E1 5947.323,E2 5947.323} C_VEL
LIN {X 0,Y 98.15,Z 803.2,A -85,B 0,C 180,E1 5935.333,E2 5935.333} C_VEL
LIN {X 0,Y 97.085,Z 799.528,A -85,B 0,C 180,E1 5924.477,E2 5924.477} C_VEL
LIN {X 0,Y 97.41,Z 795.056,A -85,B 0,C 180,E1 5914.472,E2 5914.472} C_VEL
LIN {X 0,Y 99.433,Z 789.368,A -85,B 0,C 180,E1 5904.333,E2 5904.333} C_VEL
LIN {X 0,Y 104.378,Z 781.194,A -85,B 0,C 180,E1 5893.292,E2 5893.292} C_VEL
LIN {X 0,Y 111.809,Z 771.539,A -85,B 0,C 180,E1 5883.678,E2 5883.678} C_VEL
LIN {X 0,Y 121.582,Z 759.85,A -85,B 0,C 180,E1 5875.247,E2 5875.247} C_VEL
LIN {X 0,Y 132.713,Z 746.516,A -85,B 0,C 180,E1 5868.349,E2 5868.349} C_VEL
LIN {X 0,Y 144.466,Z 731.808,A -85,B 0,C 180,E1 5862.799,E2 5862.799} C_VEL
LIN {X 0,Y 157.186,Z 714.615,A -85,B 0,C 180,E1 5858.048,E2 5858.048} C_VEL
LIN {X 0,Y 169.081,Z 696.941,A -85,B 0,C 180,E1 5854.412,E2 5854.412} C_VEL
LIN {X 0,Y 180.514,Z 678.008,A -85,B 0,C 180,E1 5851.451,E2 5851.451} C_VEL
LIN {X 0,Y 191.485,Z 657.371,A -85,B 0,C 180,E1 5848.977,E2 5848.977} C_VEL
LIN {X 0,Y 201.604,Z 635.384,A -85,B 0,C 180,E1 5846.964,E2 5846.964} C_VEL
LIN {X 0,Y 210.04,Z 613.885,A -85,B 0,C 180,E1 5845.447,E2 5845.447} C_VEL
LIN {X 0,Y 217.55,Z 591.032,A -85,B 0,C 180,E1 5844.2,E2 5844.2} C_VEL
LIN {X 0,Y 224.123,Z 566.047,A -85,B 0,C 180,E1 5843.177,E2 5843.177} C_VEL
LIN {X 0,Y 229.971,Z 536.492,A -85,B 0,C 180,E1 5842.33,E2 5842.33} C_VEL
LIN {X 0,Y 241.725,Z 470.959,A -85,B 0,C 180,E1 5840.719,E2 5840.719} C_VEL
LIN {X 0,Y 235.409,Z 460.079,A -85,B 0,C 180,E1 5835.93,E2 5835.93} C_VEL
LIN {X 0,Y 230.072,Z 451.446,A -85,B 0,C 180,E1 5831.178,E2 5831.178} C_VEL
LIN {X 0,Y 226.413,Z 445.734,A -85,B 0,C 180,E1 5827.351,E2 5827.351} C_VEL
LIN {X 0,Y 224.081,Z 442.25,A -85,B 0,C 180,E1 5824.64,E2 5824.64} C_VEL
LIN {X 0,Y 221.836,Z 438.697,A -85,B 0,C 180,E1 5821.464,E2 5821.464} C_VEL
LIN {X 0,Y 219.008,Z 434.25,A -85,B 0,C 180,E1 5816.656,E2 5816.656} C_VEL
LIN {X 0,Y 216.339,Z 430.232,A -85,B 0,C 180,E1 5810.376,E2 5810.376} C_VEL
LIN {X 0,Y 215.889,Z 429.227,A -85,B 0,C 180,E1 5808.607,E2 5808.607} C_VEL
LIN {X 0,Y 214.464,Z 428.28,A -85,B 0,C 180,E1 5801.093,E2 5801.093} C_VEL
LIN {X 0,Y 214.674,Z 428.459,A -85,B 0,C 180,E1 5794.946,E2 5794.946} C_VEL
LIN {X 0,Y 216.059,Z 429.567,A -85,B 0,C 180,E1 5789.005,E2 5789.005} C_VEL
LIN {X 0,Y 218.414,Z 433.808,A -85,B 0,C 180,E1 5782.611,E2 5782.611} C_VEL
LIN {X 0,Y 219.383,Z 435.092,A -85,B 0,C 180,E1 5780.68,E2 5780.68} C_VEL
LIN {X 0,Y 222.783,Z 440.233,A -85,B 0,C 180,E1 5775.232,E2 5775.232} C_VEL
LIN {X 0,Y 226.138,Z 445.398,A -85,B 0,C 180,E1 5770.956,E2 5770.956} C_VEL
LIN {X 0,Y 229.578,Z 450.709,A -85,B 0,C 180,E1 5767.252,E2 5767.252} C_VEL
LIN {X 0,Y 233.531,Z 456.915,A -85,B 0,C 180,E1 5763.556,E2 5763.556} C_VEL
LIN {X 0,Y 238.997,Z 467.306,A -85,B 0,C 180,E1 5758.904,E2 5758.904} C_VEL
LIN {X 0,Y 243.899,Z 477.309,A -85,B 0,C 180,E1 5755.218,E2 5755.218} C_VEL
LIN {X 0,Y 224.4,Z 583.885,A -85,B 0,C 180,E1 5752.506,E2 5752.506} C_VEL
LIN {X 0,Y 218.265,Z 607.984,A -85,B 0,C 180,E1 5751.659,E2 5751.659} C_VEL
LIN {X 0,Y 210.475,Z 631.385,A -85,B 0,C 180,E1 5750.641,E2 5750.641} C_VEL
LIN {X 0,Y 201.789,Z 653.139,A -85,B 0,C 180,E1 5749.346,E2 5749.346} C_VEL
LIN {X 0,Y 192.041,Z 674.135,A -85,B 0,C 180,E1 5747.671,E2 5747.671} C_VEL
LIN {X 0,Y 180.775,Z 695.219,A -85,B 0,C 180,E1 5745.432,E2 5745.432} C_VEL
LIN {X 0,Y 169.112,Z 714.478,A -85,B 0,C 180,E1 5742.695,E2 5742.695} C_VEL
LIN {X 0,Y 157.111,Z 732.283,A -85,B 0,C 180,E1 5739.299,E2 5739.299} C_VEL
LIN {X 0,Y 145.216,Z 748.245,A -85,B 0,C 180,E1 5735.16,E2 5735.16} C_VEL
LIN {X 0,Y 133.742,Z 762.528,A -85,B 0,C 180,E1 5730.127,E2 5730.127} C_VEL
LIN {X 0,Y 122.698,Z 775.684,A -85,B 0,C 180,E1 5723.77,E2 5723.77} C_VEL
LIN {X 0,Y 112.803,Z 787.411,A -85,B 0,C 180,E1 5715.878,E2 5715.878} C_VEL
LIN {X 0,Y 105.171,Z 796.986,A -85,B 0,C 180,E1 5706.787,E2 5706.787} C_VEL
LIN {X 0,Y 99.939,Z 805.098,A -85,B 0,C 180,E1 5696.11,E2 5696.11} C_VEL
LIN {X 0,Y 99.199,Z 806.634,A -85,B 0,C 180,E1 5693.672,E2 5693.672} C_VEL
LIN {X 0,Y 97.333,Z 808.941,A -85,B 0,C 180,E1 5689.493,E2 5689.493} C_VEL
LIN {X 0,Y 93.261,Z 811.466,A -85,B 0,C 180,E1 5683.037,E2 5683.037} C_VEL
LIN {X 0,Y 90.058,Z 813.704,A -85,B 0,C 180,E1 5674.905,E2 5674.905} C_VEL
LIN {X 0,Y 89.988,Z 814.145,A -85,B 0,C 180,E1 5673.133,E2 5673.133} C_VEL
LIN {X 0,Y 89.956,Z 815.33,A -85,B 0,C 180,E1 5668.083,E2 5668.083} C_VEL
LIN {X 0,Y 89.239,Z 816.421,A -85,B 0,C 180,E1 5658.359,E2 5658.359} C_VEL
LIN {X 0,Y 91.23,Z 816.471,A -85,B 0,C 180,E1 5643.992,E2 5643.992} C_VEL
LIN {X 0,Y 99.69,Z 814.921,A -85,B 0,C 180,E1 5628.544,E2 5628.544} C_VEL
LIN {X 0,Y 117.302,Z 811.074,A -85,B 0,C 180,E1 5614.22,E2 5614.22} C_VEL
LIN {X 0,Y 118.929,Z 810.675,A -85,B 0,C 180,E1 5613.132,E2 5613.132} C_VEL
LIN {X 0,Y 102.204,Z 809.012,A -85,B 0,C 180,E1 5600.031,E2 5600.031} C_VEL
LIN {X 0,Y 92.784,Z 805.867,A -85,B 0,C 180,E1 5584.954,E2 5584.954} C_VEL
LIN {X 0,Y 89.561,Z 802.025,A -85,B 0,C 180,E1 5571.664,E2 5571.664} C_VEL
LIN {X 0,Y 89.048,Z 798.68,A -85,B 0,C 180,E1 5562.362,E2 5562.362} C_VEL
LIN {X 0,Y 89.781,Z 793.838,A -85,B 0,C 180,E1 5551.398,E2 5551.398} C_VEL
LIN {X 0,Y 93.124,Z 786.679,A -85,B 0,C 180,E1 5539.096,E2 5539.096} C_VEL
LIN {X 0,Y 99.514,Z 777.833,A -85,B 0,C 180,E1 5527.806,E2 5527.806} C_VEL
LIN {X 0,Y 108.677,Z 767.102,A -85,B 0,C 180,E1 5517.984,E2 5517.984} C_VEL
LIN {X 0,Y 119.522,Z 754.737,A -85,B 0,C 180,E1 5510.064,E2 5510.064} C_VEL
LIN {X 0,Y 131.577,Z 740.676,A -85,B 0,C 180,E1 5503.629,E2 5503.629} C_VEL
LIN {X 0,Y 144.493,Z 724.604,A -85,B 0,C 180,E1 5498.345,E2 5498.345} C_VEL
LIN {X 0,Y 156.899,Z 707.757,A -85,B 0,C 180,E1 5494.288,E2 5494.288} C_VEL
LIN {X 0,Y 168.984,Z 689.553,A -85,B 0,C 180,E1 5490.997,E2 5490.997} C_VEL
LIN {X 0,Y 181.045,Z 668.999,A -85,B 0,C 180,E1 5488.206,E2 5488.206} C_VEL
LIN {X 0,Y 191.866,Z 647.769,A -85,B 0,C 180,E1 5486.028,E2 5486.028} C_VEL
LIN {X 0,Y 201.436,Z 625.886,A -85,B 0,C 180,E1 5484.306,E2 5484.306} C_VEL
LIN {X 0,Y 209.871,Z 602.997,A -85,B 0,C 180,E1 5482.921,E2 5482.921} C_VEL
LIN {X 0,Y 217.218,Z 578.58,A -85,B 0,C 180,E1 5481.808,E2 5481.808} C_VEL
LIN {X 0,Y 223.082,Z 553.487,A -85,B 0,C 180,E1 5480.982,E2 5480.982} C_VEL
LIN {X 0,Y 237.46,Z 475.49,A -85,B 0,C 180,E1 5479.08,E2 5479.08} C_VEL
LIN {X 0,Y 232.081,Z 466.152,A -85,B 0,C 180,E1 5474.766,E2 5474.766} C_VEL
LIN {X 0,Y 227.276,Z 458.207,A -85,B 0,C 180,E1 5470.283,E2 5470.283} C_VEL
LIN {X 0,Y 223.025,Z 451.195,A -85,B 0,C 180,E1 5465.505,E2 5465.505} C_VEL
LIN {X 0,Y 219.71,Z 446.225,A -85,B 0,C 180,E1 5461.013,E2 5461.013} C_VEL
LIN {X 0,Y 217.112,Z 441.985,A -85,B 0,C 180,E1 5456.456,E2 5456.456} C_VEL
LIN {X 0,Y 214.533,Z 438.125,A -85,B 0,C 180,E1 5450.324,E2 5450.324} C_VEL
LIN {X 0,Y 214.091,Z 437.01,A -85,B 0,C 180,E1 5448.462,E2 5448.462} C_VEL
LIN {X 0,Y 212.706,Z 436.087,A -85,B 0,C 180,E1 5441.149,E2 5441.149} C_VEL
LIN {X 0,Y 212.908,Z 436.264,A -85,B 0,C 180,E1 5434.95,E2 5434.95} C_VEL
LIN {X 0,Y 214.21,Z 437.34,A -85,B 0,C 180,E1 5429.215,E2 5429.215} C_VEL
LIN {X 0,Y 216.539,Z 441.546,A -85,B 0,C 180,E1 5422.817,E2 5422.817} C_VEL
LIN {X 0,Y 217.416,Z 442.763,A -85,B 0,C 180,E1 5421.013,E2 5421.013} C_VEL
LIN {X 0,Y 220.687,Z 447.81,A -85,B 0,C 180,E1 5415.635,E2 5415.635} C_VEL
LIN {X 0,Y 223.99,Z 453.008,A -85,B 0,C 180,E1 5411.323,E2 5411.323} C_VEL
LIN {X 0,Y 227.66,Z 458.768,A -85,B 0,C 180,E1 5407.314,E2 5407.314} C_VEL
LIN {X 0,Y 231.66,Z 465.382,A -85,B 0,C 180,E1 5403.523,E2 5403.523} C_VEL
LIN {X 0,Y 237.078,Z 476.098,A -85,B 0,C 180,E1 5398.859,E2 5398.859} C_VEL
LIN {X 0,Y 239.611,Z 481.649,A -85,B 0,C 180,E1 5396.826,E2 5396.826} C_VEL
LIN {X 0,Y 220.542,Z 583.454,A -85,B 0,C 180,E1 5394.311,E2 5394.311} C_VEL
LIN {X 0,Y 214.178,Z 607.914,A -85,B 0,C 180,E1 5393.482,E2 5393.482} C_VEL
LIN {X 0,Y 205.884,Z 632.232,A -85,B 0,C 180,E1 5392.462,E2 5392.462} C_VEL
LIN {X 0,Y 196.791,Z 654.281,A -85,B 0,C 180,E1 5391.173,E2 5391.173} C_VEL
LIN {X 0,Y 186.623,Z 675.367,A -85,B 0,C 180,E1 5389.5,E2 5389.5} C_VEL
LIN {X 0,Y 175.232,Z 695.91,A -85,B 0,C 180,E1 5387.327,E2 5387.327} C_VEL
LIN {X 0,Y 162.87,Z 715.535,A -85,B 0,C 180,E1 5384.525,E2 5384.525} C_VEL
LIN {X 0,Y 150.565,Z 733.044,A -85,B 0,C 180,E1 5381.124,E2 5381.124} C_VEL
LIN {X 0,Y 137.693,Z 749.635,A -85,B 0,C 180,E1 5376.707,E2 5376.707} C_VEL
LIN {X 0,Y 125.419,Z 764.186,A -85,B 0,C 180,E1 5371.264,E2 5371.264} C_VEL
LIN {X 0,Y 114.117,Z 776.928,A -85,B 0,C 180,E1 5364.561,E2 5364.561} C_VEL
LIN {X 0,Y 104.048,Z 788.274,A -85,B 0,C 180,E1 5356.105,E2 5356.105} C_VEL
LIN {X 0,Y 96.403,Z 797.605,A -85,B 0,C 180,E1 5346.233,E2 5346.233} C_VEL
LIN {X 0,Y 91.528,Z 805.095,A -85,B 0,C 180,E1 5334.93,E2 5334.93} C_VEL
LIN {X 0,Y 89.688,Z 810.879,A -85,B 0,C 180,E1 5322.876,E2 5322.876} C_VEL
LIN {X 0,Y 89.948,Z 813.962,A -85,B 0,C 180,E1 5313.818,E2 5313.818} C_VEL
LIN {X 0,Y 89.988,Z 814.145,A -85,B 0,C 180,E1 5313.133,E2 5313.133} C_VEL
LIN {X 0,Y 89.336,Z 814.946,A -85,B 0,C 180,E1 5309.33,E2 5309.33} C_VEL
LIN {X 0,Y 87.019,Z 815.386,A -85,B 0,C 180,E1 5304.501,E2 5304.501} C_VEL
LIN {X 0,Y 81.916,Z 815.36,A -85,B 0,C 180,E1 5292.906,E2 5292.906} C_VEL
LIN {X 0,Y 81.931,Z 815.352,A -85,B 0,C 180,E1 5289.689,E2 5289.689} C_VEL
LIN {X 0,Y 87.188,Z 814.976,A -85,B 0,C 180,E1 5274.199,E2 5274.199} C_VEL
LIN {X 0,Y 102.716,Z 812.482,A -85,B 0,C 180,E1 5257.033,E2 5257.033} C_VEL
LIN {X 0,Y 108.469,Z 811.437,A -85,B 0,C 180,E1 5253.071,E2 5253.071} C_VEL
LIN {X 0,Y 91.933,Z 808.859,A -85,B 0,C 180,E1 5238.394,E2 5238.394} C_VEL
LIN {X 0,Y 83.812,Z 805.119,A -85,B 0,C 180,E1 5222.744,E2 5222.744} C_VEL
LIN {X 0,Y 81.275,Z 800.944,A -85,B 0,C 180,E1 5208.658,E2 5208.658} C_VEL
LIN {X 0,Y 81.155,Z 796.772,A -85,B 0,C 180,E1 5197.538,E2 5197.538} C_VEL
LIN {X 0,Y 82.703,Z 791.527,A -85,B 0,C 180,E1 5186.224,E2 5186.224} C_VEL
LIN {X 0,Y 87.602,Z 783.589,A -85,B 0,C 180,E1 5173.089,E2 5173.089} C_VEL
LIN {X 0,Y 95.423,Z 774.201,A -85,B 0,C 180,E1 5161.943,E2 5161.943} C_VEL
LIN {X 0,Y 105.99,Z 762.65,A -85,B 0,C 180,E1 5152.432,E2 5152.432} C_VEL
LIN {X 0,Y 117.968,Z 749.617,A -85,B 0,C 180,E1 5144.963,E2 5144.963} C_VEL
LIN {X 0,Y 131.161,Z 734.524,A -85,B 0,C 180,E1 5138.907,E2 5138.907} C_VEL
LIN {X 0,Y 143.822,Z 718.798,A -85,B 0,C 180,E1 5134.39,E2 5134.39} C_VEL
LIN {X 0,Y 156.969,Z 700.725,A -85,B 0,C 180,E1 5130.587,E2 5130.587} C_VEL
LIN {X 0,Y 169.561,Z 681.194,A -85,B 0,C 180,E1 5127.566,E2 5127.566} C_VEL
LIN {X 0,Y 181.042,Z 660.899,A -85,B 0,C 180,E1 5125.197,E2 5125.197} C_VEL
LIN {X 0,Y 191.609,Z 639.388,A -85,B 0,C 180,E1 5123.279,E2 5123.279} C_VEL
LIN {X 0,Y 201.231,Z 616.388,A -85,B 0,C 180,E1 5121.718,E2 5121.718} C_VEL
LIN {X 0,Y 209.576,Z 592.275,A -85,B 0,C 180,E1 5120.479,E2 5120.479} C_VEL
LIN {X 0,Y 216.571,Z 566.839,A -85,B 0,C 180,E1 5119.51,E2 5119.51} C_VEL
LIN {X 0,Y 223.209,Z 534.595,A -85,B 0,C 180,E1 5118.659,E2 5118.659} C_VEL
LIN {X 0,Y 233.369,Z 480.124,A -85,B 0,C 180,E1 5117.381,E2 5117.381} C_VEL
LIN {X 0,Y 228,Z 470.597,A -85,B 0,C 180,E1 5112.743,E2 5112.743} C_VEL
LIN {X 0,Y 223.135,Z 462.464,A -85,B 0,C 180,E1 5107.754,E2 5107.754} C_VEL
LIN {X 0,Y 219.86,Z 457.363,A -85,B 0,C 180,E1 5103.827,E2 5103.827} C_VEL
LIN {X 0,Y 217.597,Z 453.752,A -85,B 0,C 180,E1 5100.553,E2 5100.553} C_VEL
LIN {X 0,Y 215.131,Z 449.648,A -85,B 0,C 180,E1 5096.105,E2 5096.105} C_VEL
LIN {X 0,Y 212.667,Z 445.827,A -85,B 0,C 180,E1 5090.02,E2 5090.02} C_VEL
LIN {X 0,Y 212.238,Z 444.757,A -85,B 0,C 180,E1 5088.095,E2 5088.095} C_VEL
LIN {X 0,Y 210.918,Z 443.871,A -85,B 0,C 180,E1 5080.852,E2 5080.852} C_VEL
LIN {X 0,Y 211.187,Z 444.122,A -85,B 0,C 180,E1 5074.615,E2 5074.615} C_VEL
LIN {X 0,Y 212.365,Z 445.112,A -85,B 0,C 180,E1 5069.429,E2 5069.429} C_VEL
LIN {X 0,Y 214.635,Z 449.274,A -85,B 0,C 180,E1 5063.031,E2 5063.031} C_VEL
LIN {X 0,Y 215.518,Z 450.6,A -85,B 0,C 180,E1 5061.181,E2 5061.181} C_VEL
LIN {X 0,Y 218.573,Z 455.359,A -85,B 0,C 180,E1 5056.063,E2 5056.063} C_VEL
LIN {X 0,Y 221.768,Z 460.489,A -85,B 0,C 180,E1 5051.786,E2 5051.786} C_VEL
LIN {X 0,Y 225.494,Z 466.42,A -85,B 0,C 180,E1 5047.641,E2 5047.641} C_VEL
LIN {X 0,Y 229.14,Z 472.725,A -85,B 0,C 180,E1 5044.063,E2 5044.063} C_VEL
LIN {X 0,Y 234.28,Z 483.144,A -85,B 0,C 180,E1 5039.508,E2 5039.508} C_VEL
LIN {X 0,Y 235.492,Z 485.981,A -85,B 0,C 180,E1 5038.487,E2 5038.487} C_VEL
LIN {X 0,Y 216.908,Z 582.67,A -85,B 0,C 180,E1 5036.177,E2 5036.177} C_VEL
LIN {X 0,Y 210.415,Z 607.075,A -85,B 0,C 180,E1 5035.382,E2 5035.382} C_VEL
LIN {X 0,Y 202.403,Z 630.184,A -85,B 0,C 180,E1 5034.464,E2 5034.464} C_VEL
LIN {X 0,Y 193.293,Z 652.075,A -85,B 0,C 180,E1 5033.269,E2 5033.269} C_VEL
LIN {X 0,Y 182.888,Z 673.472,A -85,B 0,C 180,E1 5031.678,E2 5031.678} C_VEL
LIN {X 0,Y 170.813,Z 694.905,A -85,B 0,C 180,E1 5029.52,E2 5029.52} C_VEL
LIN {X 0,Y 158.138,Z 714.581,A -85,B 0,C 180,E1 5026.81,E2 5026.81} C_VEL
LIN {X 0,Y 145.504,Z 732.082,A -85,B 0,C 180,E1 5023.502,E2 5023.502} C_VEL
LIN {X 0,Y 132.31,Z 748.557,A -85,B 0,C 180,E1 5019.19,E2 5019.19} C_VEL
LIN {X 0,Y 119.204,Z 763.445,A -85,B 0,C 180,E1 5013.599,E2 5013.599} C_VEL
LIN {X 0,Y 107.491,Z 776.001,A -85,B 0,C 180,E1 5006.831,E2 5006.831} C_VEL
LIN {X 0,Y 96.839,Z 787.331,A -85,B 0,C 180,E1 4998.012,E2 4998.012} C_VEL
LIN {X 0,Y 88.712,Z 796.663,A -85,B 0,C 180,E1 4987.481,E2 4987.481} C_VEL
LIN {X 0,Y 83.642,Z 804.025,A -85,B 0,C 180,E1 4975.482,E2 4975.482} C_VEL
LIN {X 0,Y 81.781,Z 809.682,A -85,B 0,C 180,E1 4962.706,E2 4962.706} C_VEL
LIN {X 0,Y 82.121,Z 812.791,A -85,B 0,C 180,E1 4952.785,E2 4952.785} C_VEL
LIN {X 0,Y 82.066,Z 813.876,A -85,B 0,C 180,E1 4947.699,E2 4947.699} C_VEL
LIN {X 0,Y 81.368,Z 815.033,A -85,B 0,C 180,E1 4937.214,E2 4937.214} C_VEL
LIN {X 0,Y 81.931,Z 815.352,A -85,B 0,C 180,E1 4929.689,E2 4929.689} C_VEL
LIN {X 0,Y 82.094,Z 815.251,A -85,B 0,C 180,E1 4924.269,E2 4924.269} C_VEL
LIN {X 0,Y 82.587,Z 813.797,A -85,B 0,C 180,E1 4908.669,E2 4908.669} C_VEL
LIN {X 0,Y 84.618,Z 813.484,A -85,B 0,C 180,E1 4905.119,E2 4905.119} C_VEL
LIN {X 0,Y 97.925,Z 811.753,A -85,B 0,C 180,E1 4892.965,E2 4892.965} C_VEL
LIN {X 0,Y 82.113,Z 808.341,A -85,B 0,C 180,E1 4877.001,E2 4877.001} C_VEL
LIN {X 0,Y 74.906,Z 804.057,A -85,B 0,C 180,E1 4860.01,E2 4860.01} C_VEL
LIN {X 0,Y 73.159,Z 800.014,A -85,B 0,C 180,E1 4846.576,E2 4846.576} C_VEL
LIN {X 0,Y 73.398,Z 795.428,A -85,B 0,C 180,E1 4834.054,E2 4834.054} C_VEL
LIN {X 0,Y 76.277,Z 788.831,A -85,B 0,C 180,E1 4820.051,E2 4820.051} C_VEL
LIN {X 0,Y 82.599,Z 780.56,A -85,B 0,C 180,E1 4806.989,E2 4806.989} C_VEL
LIN {X 0,Y 92.251,Z 770.164,A -85,B 0,C 180,E1 4795.699,E2 4795.699} C_VEL
LIN {X 0,Y 104.096,Z 757.998,A -85,B 0,C 180,E1 4786.753,E2 4786.753} C_VEL
LIN {X 0,Y 117.165,Z 744.18,A -85,B 0,C 180,E1 4779.832,E2 4779.832} C_VEL
LIN {X 0,Y 130.383,Z 729.206,A -85,B 0,C 180,E1 4774.591,E2 4774.591} C_VEL
LIN {X 0,Y 144.464,Z 711.594,A -85,B 0,C 180,E1 4770.222,E2 4770.222} C_VEL
LIN {X 0,Y 157.931,Z 692.647,A -85,B 0,C 180,E1 4766.849,E2 4766.849} C_VEL
LIN {X 0,Y 169.785,Z 673.707,A -85,B 0,C 180,E1 4764.342,E2 4764.342} C_VEL
LIN {X 0,Y 181.104,Z 653.055,A -85,B 0,C 180,E1 4762.266,E2 4762.266} C_VEL
LIN {X 0,Y 191.998,Z 629.88,A -85,B 0,C 180,E1 4760.505,E2 4760.505} C_VEL
LIN {X 0,Y 201.17,Z 606.559,A -85,B 0,C 180,E1 4759.162,E2 4759.162} C_VEL
LIN {X 0,Y 208.81,Z 582.831,A -85,B 0,C 180,E1 4758.127,E2 4758.127} C_VEL
LIN {X 0,Y 214.938,Z 558.801,A -85,B 0,C 180,E1 4757.358,E2 4757.358} C_VEL
LIN {X 0,Y 229.349,Z 484.815,A -85,B 0,C 180,E1 4755.689,E2 4755.689} C_VEL
LIN {X 0,Y 224.152,Z 475.62,A -85,B 0,C 180,E1 4750.864,E2 4750.864} C_VEL
LIN {X 0,Y 220.196,Z 468.913,A -85,B 0,C 180,E1 4746.513,E2 4746.513} C_VEL
LIN {X 0,Y 217.544,Z 464.548,A -85,B 0,C 180,E1 4743.07,E2 4743.07} C_VEL
LIN {X 0,Y 215.389,Z 461.132,A -85,B 0,C 180,E1 4739.914,E2 4739.914} C_VEL
LIN {X 0,Y 213.107,Z 457.266,A -85,B 0,C 180,E1 4735.657,E2 4735.657} C_VEL
LIN {X 0,Y 210.798,Z 453.501,A -85,B 0,C 180,E1 4729.673,E2 4729.673} C_VEL
LIN {X 0,Y 210.42,Z 452.521,A -85,B 0,C 180,E1 4727.833,E2 4727.833} C_VEL
LIN {X 0,Y 209.159,Z 451.679,A -85,B 0,C 180,E1 4720.907,E2 4720.907} C_VEL
LIN {X 0,Y 209.421,Z 451.928,A -85,B 0,C 180,E1 4714.616,E2 4714.616} C_VEL
LIN {X 0,Y 210.533,Z 452.923,A -85,B 0,C 180,E1 4709.593,E2 4709.593} C_VEL
LIN {X 0,Y 212.598,Z 456.862,A -85,B 0,C 180,E1 4703.503,E2 4703.503} C_VEL
LIN {X 0,Y 213.533,Z 458.225,A -85,B 0,C 180,E1 4701.562,E2 4701.562} C_VEL
LIN {X 0,Y 216.553,Z 463.079,A -85,B 0,C 180,E1 4696.354,E2 4696.354} C_VEL
LIN {X 0,Y 219.589,Z 468.021,A -85,B 0,C 180,E1 4692.22,E2 4692.22} C_VEL
LIN {X 0,Y 223.831,Z 474.864,A -85,B 0,C 180,E1 4687.44,E2 4687.44} C_VEL
LIN {X 0,Y 227.084,Z 481.007,A -85,B 0,C 180,E1 4684.163,E2 4684.163} C_VEL
LIN {X 0,Y 231.419,Z 490.104,A -85,B 0,C 180,E1 4680.193,E2 4680.193} C_VEL
LIN {X 0,Y 213.252,Z 582.425,A -85,B 0,C 180,E1 4678.072,E2 4678.072} C_VEL
LIN {X 0,Y 206.684,Z 606.653,A -85,B 0,C 180,E1 4677.323,E2 4677.323} C_VEL
LIN {X 0,Y 198.342,Z 630.271,A -85,B 0,C 180,E1 4676.441,E2 4676.441} C_VEL
LIN {X 0,Y 189.093,Z 652.012,A -85,B 0,C 180,E1 4675.313,E2 4675.313} C_VEL
LIN {X 0,Y 178.358,Z 673.581,A -85,B 0,C 180,E1 4673.78,E2 4673.78} C_VEL
LIN {X 0,Y 166.188,Z 694.589,A -85,B 0,C 180,E1 4671.739,E2 4671.739} C_VEL
LIN {X 0,Y 152.938,Z 714.53,A -85,B 0,C 180,E1 4669.066,E2 4669.066} C_VEL
LIN {X 0,Y 139.771,Z 732.121,A -85,B 0,C 180,E1 4665.779,E2 4665.779} C_VEL
LIN {X 0,Y 126.2,Z 748.401,A -85,B 0,C 180,E1 4661.518,E2 4661.518} C_VEL
LIN {X 0,Y 112.602,Z 763.228,A -85,B 0,C 180,E1 4655.885,E2 4655.885} C_VEL
LIN {X 0,Y 100.375,Z 775.694,A -85,B 0,C 180,E1 4648.932,E2 4648.932} C_VEL
LIN {X 0,Y 88.651,Z 787.485,A -85,B 0,C 180,E1 4639.073,E2 4639.073} C_VEL
LIN {X 0,Y 80.304,Z 796.587,A -85,B 0,C 180,E1 4627.587,E2 4627.587} C_VEL
LIN {X 0,Y 75.322,Z 803.736,A -85,B 0,C 180,E1 4614.291,E2 4614.291} C_VEL
LIN {X 0,Y 73.878,Z 809.176,A -85,B 0,C 180,E1 4600.126,E2 4600.126} C_VEL
LIN {X 0,Y 74.336,Z 811.746,A -85,B 0,C 180,E1 4590.763,E2 4590.763} C_VEL
LIN {X 0,Y 73.823,Z 812.862,A -85,B 0,C 180,E1 4583.772,E2 4583.772} C_VEL
LIN {X 0,Y 74.285,Z 814.075,A -85,B 0,C 180,E1 4567.852,E2 4567.852} C_VEL
LIN {X 0,Y 81.925,Z 813.741,A -85,B 0,C 180,E1 4548.764,E2 4548.764} C_VEL
LIN {X 0,Y 84.618,Z 813.484,A -85,B 0,C 180,E1 4545.119,E2 4545.119} C_VEL
LIN {X 0,Y 86.231,Z 813.165,A -85,B 0,C 180,E1 4542.129,E2 4542.129} C_VEL
LIN {X 0,Y 86.784,Z 812.596,A -85,B 0,C 180,E1 4538.457,E2 4538.457} C_VEL
LIN {X 0,Y 86.081,Z 811.799,A -85,B 0,C 180,E1 4534.239,E2 4534.239} C_VEL
LIN {X 0,Y 84.315,Z 811.039,A -85,B 0,C 180,E1 4530.679,E2 4530.679} C_VEL
LIN {X 0,Y 82.707,Z 810.605,A -85,B 0,C 180,E1 4528.799,E2 4528.799} C_VEL
LIN {X 0,Y 70.138,Z 806.361,A -85,B 0,C 180,E1 4510.691,E2 4510.691} C_VEL
LIN {X 0,Y 65.738,Z 801.895,A -85,B 0,C 180,E1 4493.9,E2 4493.9} C_VEL
LIN {X 0,Y 65.048,Z 798.277,A -85,B 0,C 180,E1 4482.109,E2 4482.109} C_VEL
LIN {X 0,Y 65.991,Z 793.458,A -85,B 0,C 180,E1 4469.007,E2 4469.007} C_VEL
LIN {X 0,Y 70.395,Z 786.195,A -85,B 0,C 180,E1 4453.6,E2 4453.6} C_VEL
LIN {X 0,Y 78.037,Z 777.603,A -85,B 0,C 180,E1 4440.839,E2 4440.839} C_VEL
LIN {X 0,Y 89.492,Z 766.329,A -85,B 0,C 180,E1 4429.59,E2 4429.59} C_VEL
LIN {X 0,Y 102.553,Z 753.577,A -85,B 0,C 180,E1 4421.25,E2 4421.25} C_VEL
LIN {X 0,Y 116.562,Z 739.105,A -85,B 0,C 180,E1 4414.926,E2 4414.926} C_VEL
LIN {X 0,Y 131.114,Z 722.47,A -85,B 0,C 180,E1 4410.004,E2 4410.004} C_VEL
LIN {X 0,Y 144.497,Z 705.415,A -85,B 0,C 180,E1 4406.433,E2 4406.433} C_VEL
LIN {X 0,Y 157.538,Z 686.733,A -85,B 0,C 180,E1 4403.557,E2 4403.557} C_VEL
LIN {X 0,Y 170.434,Z 665.633,A -85,B 0,C 180,E1 4401.157,E2 4401.157} C_VEL
LIN {X 0,Y 181.757,Z 644.173,A -85,B 0,C 180,E1 4399.324,E2 4399.324} C_VEL
LIN {X 0,Y 191.669,Z 622.183,A -85,B 0,C 180,E1 4397.892,E2 4397.892} C_VEL
LIN {X 0,Y 200.444,Z 598.903,A -85,B 0,C 180,E1 4396.738,E2 4396.738} C_VEL
LIN {X 0,Y 207.994,Z 574.039,A -85,B 0,C 180,E1 4395.824,E2 4395.824} C_VEL
LIN {X 0,Y 213.909,Z 548.407,A -85,B 0,C 180,E1 4395.155,E2 4395.155} C_VEL
LIN {X 0,Y 225.422,Z 489.604,A -85,B 0,C 180,E1 4393.909,E2 4393.909} C_VEL
LIN {X 0,Y 220.672,Z 481.008,A -85,B 0,C 180,E1 4389.168,E2 4389.168} C_VEL
LIN {X 0,Y 216.389,Z 473.518,A -85,B 0,C 180,E1 4383.966,E2 4383.966} C_VEL
LIN {X 0,Y 213.312,Z 468.657,A -85,B 0,C 180,E1 4379.435,E2 4379.435} C_VEL
LIN {X 0,Y 211.193,Z 464.972,A -85,B 0,C 180,E1 4375.385,E2 4375.385} C_VEL
LIN {X 0,Y 208.899,Z 461.031,A -85,B 0,C 180,E1 4369.126,E2 4369.126} C_VEL
LIN {X 0,Y 208.549,Z 460.26,A -85,B 0,C 180,E1 4367.472,E2 4367.472} C_VEL
LIN {X 0,Y 207.365,Z 459.446,A -85,B 0,C 180,E1 4360.379,E2 4360.379} C_VEL
LIN {X 0,Y 207.768,Z 459.838,A -85,B 0,C 180,E1 4353.928,E2 4353.928} C_VEL
LIN {X 0,Y 208.679,Z 460.654,A -85,B 0,C 180,E1 4349.868,E2 4349.868} C_VEL
LIN {X 0,Y 210.671,Z 464.558,A -85,B 0,C 180,E1 4343.787,E2 4343.787} C_VEL
LIN {X 0,Y 211.632,Z 466.027,A -85,B 0,C 180,E1 4341.765,E2 4341.765} C_VEL
LIN {X 0,Y 214.454,Z 470.625,A -85,B 0,C 180,E1 4336.798,E2 4336.798} C_VEL
LIN {X 0,Y 217.454,Z 475.618,A -85,B 0,C 180,E1 4332.612,E2 4332.612} C_VEL
LIN {X 0,Y 221.45,Z 482.238,A -85,B 0,C 180,E1 4327.977,E2 4327.977} C_VEL
LIN {X 0,Y 224.534,Z 488.309,A -85,B 0,C 180,E1 4324.722,E2 4324.722} C_VEL
LIN {X 0,Y 227.431,Z 494.666,A -85,B 0,C 180,E1 4321.939,E2 4321.939} C_VEL
LIN {X 0,Y 209.958,Z 581.671,A -85,B 0,C 180,E1 4320.045,E2 4320.045} C_VEL
LIN {X 0,Y 203.296,Z 605.742,A -85,B 0,C 180,E1 4319.34,E2 4319.34} C_VEL
LIN {X 0,Y 194.855,Z 629.235,A -85,B 0,C 180,E1 4318.526,E2 4318.526} C_VEL
LIN {X 0,Y 185.146,Z 651.622,A -85,B 0,C 180,E1 4317.441,E2 4317.441} C_VEL
LIN {X 0,Y 174.033,Z 673.412,A -85,B 0,C 180,E1 4315.972,E2 4315.972} C_VEL
LIN {X 0,Y 161.83,Z 694.014,A -85,B 0,C 180,E1 4314.075,E2 4314.075} C_VEL
LIN {X 0,Y 148.565,Z 713.548,A -85,B 0,C 180,E1 4311.59,E2 4311.59} C_VEL
LIN {X 0,Y 135.146,Z 731.044,A -85,B 0,C 180,E1 4308.472,E2 4308.472} C_VEL
LIN {X 0,Y 120.985,Z 747.522,A -85,B 0,C 180,E1 4304.302,E2 4304.302} C_VEL
LIN {X 0,Y 107.164,Z 761.968,A -85,B 0,C 180,E1 4298.893,E2 4298.893} C_VEL
LIN {X 0,Y 94.138,Z 774.602,A -85,B 0,C 180,E1 4291.817,E2 4291.817} C_VEL
LIN {X 0,Y 82.244,Z 785.844,A -85,B 0,C 180,E1 4282.193,E2 4282.193} C_VEL
LIN {X 0,Y 73.075,Z 795.104,A -85,B 0,C 180,E1 4269.969,E2 4269.969} C_VEL
LIN {X 0,Y 67.556,Z 802.341,A -85,B 0,C 180,E1 4255.408,E2 4255.408} C_VEL
LIN {X 0,Y 65.999,Z 807.778,A -85,B 0,C 180,E1 4239.97,E2 4239.97} C_VEL
LIN {X 0,Y 66.506,Z 810.294,A -85,B 0,C 180,E1 4229.991,E2 4229.991} C_VEL
LIN {X 0,Y 65.798,Z 811.493,A -85,B 0,C 180,E1 4221.08,E2 4221.08} C_VEL
LIN {X 0,Y 67.317,Z 812.698,A -85,B 0,C 180,E1 4203.044,E2 4203.044} C_VEL
LIN {X 0,Y 78.579,Z 812.393,A -85,B 0,C 180,E1 4181.336,E2 4181.336} C_VEL
LIN {X 0,Y 87.471,Z 811.594,A -85,B 0,C 180,E1 4172.925,E2 4172.925} C_VEL
LIN {X 0,Y 82.707,Z 810.605,A -85,B 0,C 180,E1 4168.799,E2 4168.799} C_VEL
LIN {X 0,Y 77.634,Z 809.629,A -85,B 0,C 180,E1 4164.67,E2 4164.67} C_VEL
LIN {X 0,Y 63.099,Z 806.03,A -85,B 0,C 180,E1 4152.264,E2 4152.264} C_VEL
LIN {X 0,Y 60.32,Z 804.651,A -85,B 0,C 180,E1 4146.751,E2 4146.751} C_VEL
LIN {X 0,Y 57.228,Z 799.764,A -85,B 0,C 180,E1 4128.116,E2 4128.116} C_VEL
LIN {X 0,Y 57.437,Z 795.074,A -85,B 0,C 180,E1 4113.105,E2 4113.105} C_VEL
LIN {X 0,Y 60.549,Z 788.959,A -85,B 0,C 180,E1 4097.406,E2 4097.406} C_VEL
LIN {X 0,Y 68.733,Z 779.773,A -85,B 0,C 180,E1 4080.901,E2 4080.901} C_VEL
LIN {X 0,Y 80.188,Z 769.143,A -85,B 0,C 180,E1 4068.658,E2 4068.658} C_VEL
LIN {X 0,Y 93.786,Z 756.579,A -85,B 0,C 180,E1 4059.605,E2 4059.605} C_VEL
LIN {X 0,Y 108.124,Z 742.481,A -85,B 0,C 180,E1 4053.07,E2 4053.07} C_VEL
LIN {X 0,Y 123.035,Z 726.418,A -85,B 0,C 180,E1 4048.078,E2 4048.078} C_VEL
LIN {X 0,Y 138.112,Z 708.208,A -85,B 0,C 180,E1 4044.187,E2 4044.187} C_VEL
LIN {X 0,Y 151.686,Z 689.586,A -85,B 0,C 180,E1 4041.352,E2 4041.352} C_VEL
LIN {X 0,Y 164.314,Z 669.778,A -85,B 0,C 180,E1 4039.13,E2 4039.13} C_VEL
LIN {X 0,Y 176.26,Z 648.118,A -85,B 0,C 180,E1 4037.315,E2 4037.315} C_VEL
LIN {X 0,Y 187.014,Z 625.133,A -85,B 0,C 180,E1 4035.866,E2 4035.866} C_VEL
LIN {X 0,Y 196.511,Z 600.649,A -85,B 0,C 180,E1 4034.709,E2 4034.709} C_VEL
LIN {X 0,Y 204.492,Z 575.002,A -85,B 0,C 180,E1 4033.821,E2 4033.821} C_VEL
LIN {X 0,Y 210.641,Z 549.049,A -85,B 0,C 180,E1 4033.183,E2 4033.183} C_VEL
LIN {X 0,Y 221.565,Z 494.42,A -85,B 0,C 180,E1 4032.065,E2 4032.065} C_VEL
LIN {X 0,Y 217.319,Z 486.664,A -85,B 0,C 180,E1 4027.482,E2 4027.482} C_VEL
LIN {X 0,Y 213.666,Z 480.186,A -85,B 0,C 180,E1 4022.707,E2 4022.707} C_VEL
LIN {X 0,Y 211.246,Z 476.175,A -85,B 0,C 180,E1 4018.939,E2 4018.939} C_VEL
LIN {X 0,Y 209.145,Z 472.539,A -85,B 0,C 180,E1 4014.827,E2 4014.827} C_VEL
LIN {X 0,Y 206.855,Z 468.109,A -85,B 0,C 180,E1 4007.685,E2 4007.685} C_VEL
LIN {X 0,Y 205.615,Z 467.269,A -85,B 0,C 180,E1 4000.657,E2 4000.657} C_VEL
LIN {X 0,Y 205.922,Z 467.578,A -85,B 0,C 180,E1 3994.373,E2 3994.373} C_VEL
LIN {X 0,Y 206.837,Z 468.427,A -85,B 0,C 180,E1 3990.091,E2 3990.091} C_VEL
LIN {X 0,Y 208.62,Z 472.108,A -85,B 0,C 180,E1 3984.337,E2 3984.337} C_VEL
LIN {X 0,Y 209.674,Z 473.681,A -85,B 0,C 180,E1 3982.126,E2 3982.126} C_VEL
LIN {X 0,Y 212.45,Z 478.34,A -85,B 0,C 180,E1 3977.102,E2 3977.102} C_VEL
LIN {X 0,Y 215.385,Z 483.382,A -85,B 0,C 180,E1 3972.871,E2 3972.871} C_VEL
LIN {X 0,Y 219.142,Z 489.816,A -85,B 0,C 180,E1 3968.392,E2 3968.392} C_VEL
LIN {X 0,Y 221.995,Z 495.584,A -85,B 0,C 180,E1 3965.307,E2 3965.307} C_VEL
LIN {X 0,Y 223.529,Z 499.174,A -85,B 0,C 180,E1 3963.737,E2 3963.737} C_VEL
LIN {X 0,Y 206.557,Z 581.485,A -85,B 0,C 180,E1 3962.037,E2 3962.037} C_VEL
LIN {X 0,Y 199.767,Z 605.58,A -85,B 0,C 180,E1 3961.382,E2 3961.382} C_VEL
LIN {X 0,Y 190.972,Z 629.605,A -85,B 0,C 180,E1 3960.619,E2 3960.619} C_VEL
LIN {X 0,Y 180.966,Z 652.159,A -85,B 0,C 180,E1 3959.6,E2 3959.6} C_VEL
LIN {X 0,Y 169.689,Z 673.738,A -85,B 0,C 180,E1 3958.235,E2 3958.235} C_VEL
LIN {X 0,Y 157.266,Z 694.187,A -85,B 0,C 180,E1 3956.459,E2 3956.459} C_VEL
LIN {X 0,Y 143.726,Z 713.515,A -85,B 0,C 180,E1 3954.111,E2 3954.111} C_VEL
LIN {X 0,Y 129.555,Z 731.329,A -85,B 0,C 180,E1 3951.03,E2 3951.03} C_VEL
LIN {X 0,Y 115.834,Z 746.713,A -85,B 0,C 180,E1 3947.239,E2 3947.239} C_VEL
LIN {X 0,Y 101.049,Z 761.558,A -85,B 0,C 180,E1 3941.767,E2 3941.767} C_VEL
LIN {X 0,Y 87.416,Z 774.129,A -85,B 0,C 180,E1 3934.618,E2 3934.618} C_VEL
LIN {X 0,Y 74.851,Z 785.293,A -85,B 0,C 180,E1 3924.557,E2 3924.557} C_VEL
LIN {X 0,Y 65.059,Z 794.512,A -85,B 0,C 180,E1 3911.128,E2 3911.128} C_VEL
LIN {X 0,Y 59.359,Z 801.702,A -85,B 0,C 180,E1 3894.523,E2 3894.523} C_VEL
LIN {X 0,Y 58.181,Z 806.787,A -85,B 0,C 180,E1 3877.892,E2 3877.892} C_VEL
LIN {X 0,Y 58.663,Z 808.714,A -85,B 0,C 180,E1 3869.014,E2 3869.014} C_VEL
LIN {X 0,Y 57.882,Z 810.214,A -85,B 0,C 180,E1 3855.995,E2 3855.995} C_VEL
LIN {X 0,Y 61.532,Z 811.336,A -85,B 0,C 180,E1 3835.328,E2 3835.328} C_VEL
LIN {X 0,Y 77.078,Z 810.985,A -85,B 0,C 180,E1 3812.953,E2 3812.953} C_VEL
LIN {X 0,Y 62.573,Z 806.1,A -85,B 0,C 180,E1 3792.939,E2 3792.939} C_VEL
LIN {X 0,Y 60.32,Z 804.651,A -85,B 0,C 180,E1 3786.751,E2 3786.751} C_VEL
LIN {X 0,Y 57.815,Z 803.016,A -85,B 0,C 180,E1 3780.388,E2 3780.388} C_VEL
LIN {X 0,Y 53.339,Z 800.215,A -85,B 0,C 180,E1 3770.865,E2 3770.865} C_VEL
LIN {X 0,Y 49.45,Z 795.991,A -85,B 0,C 180,E1 3756.355,E2 3756.355} C_VEL
LIN {X 0,Y 49.505,Z 794.67,A -85,B 0,C 180,E1 3752.011,E2 3752.011} C_VEL
LIN {X 0,Y 54.051,Z 787.341,A -85,B 0,C 180,E1 3731.768,E2 3731.768} C_VEL
LIN {X 0,Y 62.512,Z 778.996,A -85,B 0,C 180,E1 3716.432,E2 3716.432} C_VEL
LIN {X 0,Y 75.382,Z 767.822,A -85,B 0,C 180,E1 3703.82,E2 3703.82} C_VEL
LIN {X 0,Y 89.969,Z 755.021,A -85,B 0,C 180,E1 3695.107,E2 3695.107} C_VEL
LIN {X 0,Y 105.279,Z 740.518,A -85,B 0,C 180,E1 3688.917,E2 3688.917} C_VEL
LIN {X 0,Y 120.911,Z 723.862,A -85,B 0,C 180,E1 3684.31,E2 3684.31} C_VEL
LIN {X 0,Y 135.113,Z 706.809,A -85,B 0,C 180,E1 3681.064,E2 3681.064} C_VEL
LIN {X 0,Y 149.304,Z 687.456,A -85,B 0,C 180,E1 3678.414,E2 3678.414} C_VEL
LIN {X 0,Y 162.555,Z 666.671,A -85,B 0,C 180,E1 3676.344,E2 3676.344} C_VEL
LIN {X 0,Y 174.53,Z 644.823,A -85,B 0,C 180,E1 3674.724,E2 3674.724} C_VEL
LIN {X 0,Y 184.542,Z 623.417,A -85,B 0,C 180,E1 3673.516,E2 3673.516} C_VEL
LIN {X 0,Y 193.642,Z 600.049,A -85,B 0,C 180,E1 3672.517,E2 3672.517} C_VEL
LIN {X 0,Y 201.479,Z 575.048,A -85,B 0,C 180,E1 3671.728,E2 3671.728} C_VEL
LIN {X 0,Y 207.654,Z 549.296,A -85,B 0,C 180,E1 3671.149,E2 3671.149} C_VEL
LIN {X 0,Y 217.814,Z 499.285,A -85,B 0,C 180,E1 3670.188,E2 3670.188} C_VEL
LIN {X 0,Y 213.875,Z 491.955,A -85,B 0,C 180,E1 3665.578,E2 3665.578} C_VEL
LIN {X 0,Y 210.999,Z 486.94,A -85,B 0,C 180,E1 3661.563,E2 3661.563} C_VEL
LIN {X 0,Y 209.094,Z 483.548,A -85,B 0,C 180,E1 3658.268,E2 3658.268} C_VEL
LIN {X 0,Y 207.273,Z 480.274,A -85,B 0,C 180,E1 3654.602,E2 3654.602} C_VEL
LIN {X 0,Y 204.964,Z 475.843,A -85,B 0,C 180,E1 3647.311,E2 3647.311} C_VEL
LIN {X 0,Y 203.837,Z 475.052,A -85,B 0,C 180,E1 3640.346,E2 3640.346} C_VEL
LIN {X 0,Y 204.233,Z 475.448,A -85,B 0,C 180,E1 3633.919,E2 3633.919} C_VEL
LIN {X 0,Y 204.998,Z 476.202,A -85,B 0,C 180,E1 3630.318,E2 3630.318} C_VEL
LIN {X 0,Y 206.869,Z 480.007,A -85,B 0,C 180,E1 3624.252,E2 3624.252} C_VEL
LIN {X 0,Y 208.095,Z 482.183,A -85,B 0,C 180,E1 3621.561,E2 3621.561} C_VEL
LIN {X 0,Y 210.329,Z 485.867,A -85,B 0,C 180,E1 3617.565,E2 3617.565} C_VEL
LIN {X 0,Y 213.187,Z 490.944,A -85,B 0,C 180,E1 3613.282,E2 3613.282} C_VEL
LIN {X 0,Y 216.773,Z 497.268,A -85,B 0,C 180,E1 3608.885,E2 3608.885} C_VEL
LIN {X 0,Y 219.634,Z 503.177,A -85,B 0,C 180,E1 3605.744,E2 3605.744} C_VEL
LIN {X 0,Y 219.717,Z 503.795,A -85,B 0,C 180,E1 3605.583,E2 3605.583} C_VEL
LIN {X 0,Y 203.479,Z 581.051,A -85,B 0,C 180,E1 3604.099,E2 3604.099} C_VEL
LIN {X 0,Y 196.527,Z 605.319,A -85,B 0,C 180,E1 3603.496,E2 3603.496} C_VEL
LIN {X 0,Y 188.195,Z 627.76,A -85,B 0,C 180,E1 3602.86,E2 3602.86} C_VEL
LIN {X 0,Y 178.571,Z 649.32,A -85,B 0,C 180,E1 3602.001,E2 3602.001} C_VEL
LIN {X 0,Y 166.979,Z 671.393,A -85,B 0,C 180,E1 3600.764,E2 3600.764} C_VEL
LIN {X 0,Y 153.985,Z 692.54,A -85,B 0,C 180,E1 3599.109,E2 3599.109} C_VEL
LIN {X 0,Y 140.165,Z 712.005,A -85,B 0,C 180,E1 3596.963,E2 3596.963} C_VEL
LIN {X 0,Y 126.111,Z 729.399,A -85,B 0,C 180,E1 3594.224,E2 3594.224} C_VEL
LIN {X 0,Y 111.179,Z 745.707,A -85,B 0,C 180,E1 3590.486,E2 3590.486} C_VEL
LIN {X 0,Y 96.812,Z 759.611,A -85,B 0,C 180,E1 3585.641,E2 3585.641} C_VEL
LIN {X 0,Y 81.745,Z 772.872,A -85,B 0,C 180,E1 3578.351,E2 3578.351} C_VEL
LIN {X 0,Y 68.296,Z 784.07,A -85,B 0,C 180,E1 3568.099,E2 3568.099} C_VEL
LIN {X 0,Y 57.717,Z 793.232,A -85,B 0,C 180,E1 3553.849,E2 3553.849} C_VEL
LIN {X 0,Y 51.488,Z 800.421,A -85,B 0,C 180,E1 3535.279,E2 3535.279} C_VEL
LIN {X 0,Y 50.375,Z 805.319,A -85,B 0,C 180,E1 3516.828,E2 3516.828} C_VEL
LIN {X 0,Y 50.847,Z 806.932,A -85,B 0,C 180,E1 3508.862,E2 3508.862} C_VEL
LIN {X 0,Y 50.27,Z 808.702,A -85,B 0,C 180,E1 3491.432,E2 3491.432} C_VEL
LIN {X 0,Y 56.336,Z 809.878,A -85,B 0,C 180,E1 3467.577,E2 3467.577} C_VEL
LIN {X 0,Y 66.647,Z 809.939,A -85,B 0,C 180,E1 3452.977,E2 3452.977} C_VEL
LIN {X 0,Y 52.895,Z 804.372,A -85,B 0,C 180,E1 3429.81,E2 3429.81} C_VEL
LIN {X 0,Y 49.378,Z 799.818,A -85,B 0,C 180,E1 3410.693,E2 3410.693} C_VEL
LIN {X 0,Y 49.284,Z 795.507,A -85,B 0,C 180,E1 3394.801,E2 3394.801} C_VEL
LIN {X 0,Y 49.505,Z 794.67,A -85,B 0,C 180,E1 3392.011,E2 3392.011} C_VEL
LIN {X 0,Y 49.72,Z 792.412,A -85,B 0,C 180,E1 3384.809,E2 3384.809} C_VEL
LIN {X 0,Y 49.417,Z 788.282,A -85,B 0,C 180,E1 3372.797,E2 3372.797} C_VEL
LIN {X 0,Y 51.187,Z 783.227,A -85,B 0,C 180,E1 3360.026,E2 3360.026} C_VEL
LIN {X 0,Y 53.576,Z 780.689,A -85,B 0,C 180,E1 3355.183,E2 3355.183} C_VEL
LIN {X 0,Y 67.241,Z 769.648,A -85,B 0,C 180,E1 3341.134,E2 3341.134} C_VEL
LIN {X 0,Y 82.041,Z 757.461,A -85,B 0,C 180,E1 3332.342,E2 3332.342} C_VEL
LIN {X 0,Y 97.684,Z 743.323,A -85,B 0,C 180,E1 3326.214,E2 3326.214} C_VEL
LIN {X 0,Y 113.104,Z 727.81,A -85,B 0,C 180,E1 3321.871,E2 3321.871} C_VEL
LIN {X 0,Y 128.526,Z 710.289,A -85,B 0,C 180,E1 3318.545,E2 3318.545} C_VEL
LIN {X 0,Y 142.211,Z 692.579,A -85,B 0,C 180,E1 3316.174,E2 3316.174} C_VEL
LIN {X 0,Y 155.858,Z 672.273,A -85,B 0,C 180,E1 3314.189,E2 3314.189} C_VEL
LIN {X 0,Y 168.684,Z 650.022,A -85,B 0,C 180,E1 3312.594,E2 3312.594} C_VEL
LIN {X 0,Y 180.172,Z 626.403,A -85,B 0,C 180,E1 3311.337,E2 3311.337} C_VEL
LIN {X 0,Y 190.007,Z 601.935,A -85,B 0,C 180,E1 3310.364,E2 3310.364} C_VEL
LIN {X 0,Y 198.259,Z 576.371,A -85,B 0,C 180,E1 3309.618,E2 3309.618} C_VEL
LIN {X 0,Y 204.668,Z 550.38,A -85,B 0,C 180,E1 3309.082,E2 3309.082} C_VEL
LIN {X 0,Y 214.278,Z 504.437,A -85,B 0,C 180,E1 3308.296,E2 3308.296} C_VEL
LIN {X 0,Y 210.651,Z 497.623,A -85,B 0,C 180,E1 3303.672,E2 3303.672} C_VEL
LIN {X 0,Y 207.585,Z 491.943,A -85,B 0,C 180,E1 3298.82,E2 3298.82} C_VEL
LIN {X 0,Y 205.209,Z 487.801,A -85,B 0,C 180,E1 3293.972,E2 3293.972} C_VEL
LIN {X 0,Y 203.146,Z 483.621,A -85,B 0,C 180,E1 3287.162,E2 3287.162} C_VEL
LIN {X 0,Y 202.075,Z 482.858,A -85,B 0,C 180,E1 3280.366,E2 3280.366} C_VEL
LIN {X 0,Y 202.465,Z 483.253,A -85,B 0,C 180,E1 3273.915,E2 3273.915} C_VEL
LIN {X 0,Y 203.162,Z 483.979,A -85,B 0,C 180,E1 3270.549,E2 3270.549} C_VEL
LIN {X 0,Y 205.119,Z 487.902,A -85,B 0,C 180,E1 3264.166,E2 3264.166} C_VEL
LIN {X 0,Y 208.082,Z 493.2,A -85,B 0,C 180,E1 3258.195,E2 3258.195} C_VEL
LIN {X 0,Y 210.896,Z 498.331,A -85,B 0,C 180,E1 3253.834,E2 3253.834} C_VEL
LIN {X 0,Y 214.42,Z 504.717,A -85,B 0,C 180,E1 3249.389,E2 3249.389} C_VEL
LIN {X 0,Y 216.07,Z 508.303,A -85,B 0,C 180,E1 3247.486,E2 3247.486} C_VEL
LIN {X 0,Y 200.539,Z 580.517,A -85,B 0,C 180,E1 3246.207,E2 3246.207} C_VEL
LIN {X 0,Y 193.402,Z 604.926,A -85,B 0,C 180,E1 3245.658,E2 3245.658} C_VEL
LIN {X 0,Y 184.177,Z 629.262,A -85,B 0,C 180,E1 3245.05,E2 3245.05} C_VEL
LIN {X 0,Y 173.428,Z 652.563,A -85,B 0,C 180,E1 3244.196,E2 3244.196} C_VEL
LIN {X 0,Y 161.188,Z 674.882,A -85,B 0,C 180,E1 3243.015,E2 3243.015} C_VEL
LIN {X 0,Y 148.017,Z 695.373,A -85,B 0,C 180,E1 3241.494,E2 3241.494} C_VEL
LIN {X 0,Y 134.455,Z 713.657,A -85,B 0,C 180,E1 3239.568,E2 3239.568} C_VEL
LIN {X 0,Y 119.158,Z 731.671,A -85,B 0,C 180,E1 3236.798,E2 3236.798} C_VEL
LIN {X 0,Y 103.716,Z 747.607,A -85,B 0,C 180,E1 3233.141,E2 3233.141} C_VEL
LIN {X 0,Y 88.827,Z 761.315,A -85,B 0,C 180,E1 3228.285,E2 3228.285} C_VEL
LIN {X 0,Y 73.585,Z 773.873,A -85,B 0,C 180,E1 3220.957,E2 3220.957} C_VEL
LIN {X 0,Y 59.891,Z 784.445,A -85,B 0,C 180,E1 3210.221,E2 3210.221} C_VEL
LIN {X 0,Y 48.913,Z 793.333,A -85,B 0,C 180,E1 3194.011,E2 3194.011} C_VEL
LIN {X 0,Y 43.178,Z 799.892,A -85,B 0,C 180,E1 3173.168,E2 3173.168} C_VEL
LIN {X 0,Y 42.676,Z 804.094,A -85,B 0,C 180,E1 3154.017,E2 3154.017} C_VEL
LIN {X 0,Y 43.021,Z 805.116,A -85,B 0,C 180,E1 3148.49,E2 3148.49} C_VEL
LIN {X 0,Y 43.24,Z 807.221,A -85,B 0,C 180,E1 3123.924,E2 3123.924} C_VEL
LIN {X 0,Y 54.857,Z 808.448,A -85,B 0,C 180,E1 3094.879,E2 3094.879} C_VEL
LIN {X 0,Y 56.162,Z 808.441,A -85,B 0,C 180,E1 3092.964,E2 3092.964} C_VEL
LIN {X 0,Y 43.916,Z 802.782,A -85,B 0,C 180,E1 3067.869,E2 3067.869} C_VEL
LIN {X 0,Y 41.14,Z 798.002,A -85,B 0,C 180,E1 3045.954,E2 3045.954} C_VEL
LIN {X 0,Y 42.233,Z 792.736,A -85,B 0,C 180,E1 3025.399,E2 3025.399} C_VEL
LIN {X 0,Y 47.842,Z 785.817,A -85,B 0,C 180,E1 3005.436,E2 3005.436} C_VEL
LIN {X 0,Y 53.576,Z 780.689,A -85,B 0,C 180,E1 2995.183,E2 2995.183} C_VEL
LIN {X 0,Y 57.115,Z 777.136,A -85,B 0,C 180,E1 2989.078,E2 2989.078} C_VEL
LIN {X 0,Y 66.125,Z 766.549,A -85,B 0,C 180,E1 2973.988,E2 2973.988} C_VEL
LIN {X 0,Y 70.341,Z 762.834,A -85,B 0,C 180,E1 2970.907,E2 2970.907} C_VEL
LIN {X 0,Y 86.399,Z 749.622,A -85,B 0,C 180,E1 2964.301,E2 2964.301} C_VEL
LIN {X 0,Y 102.133,Z 735.01,A -85,B 0,C 180,E1 2959.856,E2 2959.856} C_VEL
LIN {X 0,Y 117.68,Z 718.647,A -85,B 0,C 180,E1 2956.58,E2 2956.58} C_VEL
LIN {X 0,Y 133.105,Z 700.124,A -85,B 0,C 180,E1 2954.026,E2 2954.026} C_VEL
LIN {X 0,Y 147.052,Z 680.891,A -85,B 0,C 180,E1 2952.138,E2 2952.138} C_VEL
LIN {X 0,Y 160.01,Z 660.255,A -85,B 0,C 180,E1 2950.639,E2 2950.639} C_VEL
LIN {X 0,Y 171.916,Z 638.033,A -85,B 0,C 180,E1 2949.435,E2 2949.435} C_VEL
LIN {X 0,Y 182.579,Z 614.171,A -85,B 0,C 180,E1 2948.478,E2 2948.478} C_VEL
LIN {X 0,Y 191.676,Z 589.182,A -85,B 0,C 180,E1 2947.727,E2 2947.727} C_VEL
LIN {X 0,Y 198.971,Z 563.684,A -85,B 0,C 180,E1 2947.166,E2 2947.166} C_VEL
LIN {X 0,Y 210.639,Z 509.45,A -85,B 0,C 180,E1 2946.278,E2 2946.278} C_VEL
LIN {X 0,Y 207.377,Z 503.065,A -85,B 0,C 180,E1 2941.65,E2 2941.65} C_VEL
LIN {X 0,Y 204.933,Z 498.673,A -85,B 0,C 180,E1 2937.396,E2 2937.396} C_VEL
LIN {X 0,Y 203.329,Z 495.535,A -85,B 0,C 180,E1 2933.743,E2 2933.743} C_VEL
LIN {X 0,Y 201.279,Z 491.377,A -85,B 0,C 180,E1 2926.898,E2 2926.898} C_VEL
LIN {X 0,Y 200.285,Z 490.638,A -85,B 0,C 180,E1 2920.084,E2 2920.084} C_VEL
LIN {X 0,Y 200.834,Z 491.149,A -85,B 0,C 180,E1 2913.2,E2 2913.2} C_VEL
LIN {X 0,Y 201.321,Z 491.767,A -85,B 0,C 180,E1 2910.762,E2 2910.762} C_VEL
LIN {X 0,Y 203.639,Z 496.501,A -85,B 0,C 180,E1 2903.35,E2 2903.35} C_VEL
LIN {X 0,Y 206.028,Z 500.883,A -85,B 0,C 180,E1 2898.53,E2 2898.53} C_VEL
LIN {X 0,Y 208.605,Z 505.681,A -85,B 0,C 180,E1 2894.428,E2 2894.428} C_VEL
LIN {X 0,Y 212.318,Z 512.625,A -85,B 0,C 180,E1 2889.62,E2 2889.62} C_VEL
LIN {X 0,Y 212.407,Z 513.23,A -85,B 0,C 180,E1 2889.431,E2 2889.431} C_VEL
LIN {X 0,Y 197.77,Z 580.104,A -85,B 0,C 180,E1 2888.364,E2 2888.364} C_VEL
LIN {X 0,Y 190.77,Z 603.825,A -85,B 0,C 180,E1 2887.897,E2 2887.897} C_VEL
LIN {X 0,Y 181.47,Z 628.227,A -85,B 0,C 180,E1 2887.392,E2 2887.392} C_VEL
LIN {X 0,Y 171.092,Z 650.534,A -85,B 0,C 180,E1 2886.707,E2 2886.707} C_VEL
LIN {X 0,Y 159.343,Z 671.861,A -85,B 0,C 180,E1 2885.757,E2 2885.757} C_VEL
LIN {X 0,Y 146.42,Z 691.974,A -85,B 0,C 180,E1 2884.505,E2 2884.505} C_VEL
LIN {X 0,Y 131.62,Z 711.848,A -85,B 0,C 180,E1 2882.736,E2 2882.736} C_VEL
LIN {X 0,Y 116.475,Z 729.508,A -85,B 0,C 180,E1 2880.404,E2 2880.404} C_VEL
LIN {X 0,Y 101.085,Z 745.215,A -85,B 0,C 180,E1 2877.318,E2 2877.318} C_VEL
LIN {X 0,Y 85.612,Z 759.031,A -85,B 0,C 180,E1 2873.019,E2 2873.019} C_VEL
LIN {X 0,Y 69.894,Z 771.482,A -85,B 0,C 180,E1 2866.56,E2 2866.56} C_VEL
LIN {X 0,Y 54.665,Z 782.548,A -85,B 0,C 180,E1 2856.113,E2 2856.113} C_VEL
LIN {X 0,Y 42.238,Z 791.575,A -85,B 0,C 180,E1 2839.223,E2 2839.223} C_VEL
LIN {X 0,Y 35.248,Z 798.609,A -85,B 0,C 180,E1 2813.381,E2 2813.381} C_VEL
LIN {X 0,Y 35.115,Z 802.805,A -85,B 0,C 180,E1 2789.984,E2 2789.984} C_VEL
LIN {X 0,Y 34.965,Z 803.392,A -85,B 0,C 180,E1 2785.063,E2 2785.063} C_VEL
LIN {X 0,Y 37.57,Z 805.689,A -85,B 0,C 180,E1 2752.24,E2 2752.24} C_VEL
LIN {X 0,Y 45.77,Z 806.533,A -85,B 0,C 180,E1 2733.121,E2 2733.121} C_VEL
LIN {X 0,Y 35.26,Z 801.046,A -85,B 0,C 180,E1 2706.535,E2 2706.535} C_VEL
LIN {X 0,Y 33.118,Z 796.854,A -85,B 0,C 180,E1 2684.258,E2 2684.258} C_VEL
LIN {X 0,Y 34.762,Z 791.715,A -85,B 0,C 180,E1 2660.773,E2 2660.773} C_VEL
LIN {X 0,Y 43.266,Z 783.439,A -85,B 0,C 180,E1 2635.719,E2 2635.719} C_VEL
LIN {X 0,Y 56.025,Z 773.754,A -85,B 0,C 180,E1 2620.291,E2 2620.291} C_VEL
LIN {X 0,Y 70.341,Z 762.834,A -85,B 0,C 180,E1 2610.907,E2 2610.907} C_VEL
LIN {X 0,Y 75.261,Z 758.484,A -85,B 0,C 180,E1 2607.702,E2 2607.702} C_VEL
LIN {X 0,Y 87.05,Z 745.815,A -85,B 0,C 180,E1 2598.879,E2 2598.879} C_VEL
LIN {X 0,Y 91.484,Z 741.484,A -85,B 0,C 180,E1 2597.283,E2 2597.283} C_VEL
LIN {X 0,Y 108.399,Z 725.06,A -85,B 0,C 180,E1 2593.941,E2 2593.941} C_VEL
LIN {X 0,Y 123.684,Z 707.956,A -85,B 0,C 180,E1 2591.628,E2 2591.628} C_VEL
LIN {X 0,Y 138.471,Z 688.894,A -85,B 0,C 180,E1 2589.813,E2 2589.813} C_VEL
LIN {X 0,Y 152.105,Z 668.582,A -85,B 0,C 180,E1 2588.405,E2 2588.405} C_VEL
LIN {X 0,Y 164.751,Z 646.597,A -85,B 0,C 180,E1 2587.275,E2 2587.275} C_VEL
LIN {X 0,Y 175.644,Z 624.22,A -85,B 0,C 180,E1 2586.405,E2 2586.405} C_VEL
LIN {X 0,Y 185.093,Z 600.906,A -85,B 0,C 180,E1 2585.717,E2 2585.717} C_VEL
LIN {X 0,Y 193.159,Z 576.28,A -85,B 0,C 180,E1 2585.176,E2 2585.176} C_VEL
LIN {X 0,Y 199.656,Z 550.52,A -85,B 0,C 180,E1 2584.774,E2 2584.774} C_VEL
LIN {X 0,Y 207.347,Z 514.749,A -85,B 0,C 180,E1 2584.282,E2 2584.282} C_VEL
LIN {X 0,Y 204.486,Z 509.264,A -85,B 0,C 180,E1 2579.926,E2 2579.926} C_VEL
LIN {X 0,Y 202.631,Z 505.839,A -85,B 0,C 180,E1 2576.494,E2 2576.494} C_VEL
LIN {X 0,Y 201.26,Z 503.054,A -85,B 0,C 180,E1 2573.107,E2 2573.107} C_VEL
LIN {X 0,Y 199.412,Z 499.133,A -85,B 0,C 180,E1 2566.618,E2 2566.618} C_VEL
LIN {X 0,Y 198.497,Z 498.419,A -85,B 0,C 180,E1 2559.765,E2 2559.765} C_VEL
LIN {X 0,Y 199.227,Z 499.051,A -85,B 0,C 180,E1 2552.474,E2 2552.474} C_VEL
LIN {X 0,Y 199.508,Z 499.724,A -85,B 0,C 180,E1 2550.738,E2 2550.738} C_VEL
LIN {X 0,Y 201.605,Z 504.045,A -85,B 0,C 180,E1 2543.836,E2 2543.836} C_VEL
LIN {X 0,Y 203.963,Z 508.526,A -85,B 0,C 180,E1 2538.906,E2 2538.906} C_VEL
LIN {X 0,Y 206.498,Z 513.343,A -85,B 0,C 180,E1 2534.787,E2 2534.787} C_VEL
LIN {X 0,Y 208.95,Z 518.141,A -85,B 0,C 180,E1 2531.437,E2 2531.437} C_VEL
LIN {X 0,Y 195.221,Z 579.631,A -85,B 0,C 180,E1 2530.572,E2 2530.572} C_VEL
LIN {X 0,Y 188.172,Z 603.121,A -85,B 0,C 180,E1 2530.176,E2 2530.176} C_VEL
LIN {X 0,Y 179.07,Z 626.716,A -85,B 0,C 180,E1 2529.788,E2 2529.788} C_VEL
LIN {X 0,Y 168.603,Z 649.102,A -85,B 0,C 180,E1 2529.242,E2 2529.242} C_VEL
LIN {X 0,Y 156.672,Z 670.66,A -85,B 0,C 180,E1 2528.463,E2 2528.463} C_VEL
LIN {X 0,Y 143.159,Z 691.483,A -85,B 0,C 180,E1 2527.395,E2 2527.395} C_VEL
LIN {X 0,Y 128.153,Z 711.323,A -85,B 0,C 180,E1 2525.916,E2 2525.916} C_VEL
LIN {X 0,Y 112.739,Z 728.869,A -85,B 0,C 180,E1 2523.936,E2 2523.936} C_VEL
LIN {X 0,Y 97,Z 744.47,A -85,B 0,C 180,E1 2521.291,E2 2521.291} C_VEL
LIN {X 0,Y 80.069,Z 759.04,A -85,B 0,C 180,E1 2517.26,E2 2517.26} C_VEL
LIN {X 0,Y 63.714,Z 771.344,A -85,B 0,C 180,E1 2511.294,E2 2511.294} C_VEL
LIN {X 0,Y 47.575,Z 782.213,A -85,B 0,C 180,E1 2501.001,E2 2501.001} C_VEL
LIN {X 0,Y 34.113,Z 791.065,A -85,B 0,C 180,E1 2482.287,E2 2482.287} C_VEL
LIN {X 0,Y 27.011,Z 797.955,A -85,B 0,C 180,E1 2449.438,E2 2449.438} C_VEL
LIN {X 0,Y 27.367,Z 801.055,A -85,B 0,C 180,E1 2426.838,E2 2426.838} C_VEL
LIN {X 0,Y 30.145,Z 803.424,A -85,B 0,C 180,E1 2388.419,E2 2388.419} C_VEL
LIN {X 0,Y 35.531,Z 804.244,A -85,B 0,C 180,E1 2373.717,E2 2373.717} C_VEL
LIN {X 0,Y 26.306,Z 798.743,A -85,B 0,C 180,E1 2342.208,E2 2342.208} C_VEL
LIN {X 0,Y 25.281,Z 794.406,A -85,B 0,C 180,E1 2314.246,E2 2314.246} C_VEL
LIN {X 0,Y 30.108,Z 788.202,A -85,B 0,C 180,E1 2283.925,E2 2283.925} C_VEL
LIN {X 0,Y 42.766,Z 778.995,A -85,B 0,C 180,E1 2261.002,E2 2261.002} C_VEL
LIN {X 0,Y 58.994,Z 767.687,A -85,B 0,C 180,E1 2248.622,E2 2248.622} C_VEL
LIN {X 0,Y 75.79,Z 754.874,A -85,B 0,C 180,E1 2241.586,E2 2241.586} C_VEL
LIN {X 0,Y 91.484,Z 741.484,A -85,B 0,C 180,E1 2237.283,E2 2237.283} C_VEL
LIN {X 0,Y 96.504,Z 736.397,A -85,B 0,C 180,E1 2235.559,E2 2235.559} C_VEL
LIN {X 0,Y 108.482,Z 721.925,A -85,B 0,C 180,E1 2229.96,E2 2229.96} C_VEL
LIN {X 0,Y 112.774,Z 717.044,A -85,B 0,C 180,E1 2229.026,E2 2229.026} C_VEL
LIN {X 0,Y 128.372,Z 698.608,A -85,B 0,C 180,E1 2227.345,E2 2227.345} C_VEL
LIN {X 0,Y 142.857,Z 678.828,A -85,B 0,C 180,E1 2226.054,E2 2226.054} C_VEL
LIN {X 0,Y 156.247,Z 657.524,A -85,B 0,C 180,E1 2225.021,E2 2225.021} C_VEL
LIN {X 0,Y 168.489,Z 634.436,A -85,B 0,C 180,E1 2224.194,E2 2224.194} C_VEL
LIN {X 0,Y 178.847,Z 611.015,A -85,B 0,C 180,E1 2223.563,E2 2223.563} C_VEL
LIN {X 0,Y 187.584,Z 586.824,A -85,B 0,C 180,E1 2223.063,E2 2223.063} C_VEL
LIN {X 0,Y 194.544,Z 562.47,A -85,B 0,C 180,E1 2222.694,E2 2222.694} C_VEL
LIN {X 0,Y 203.97,Z 520.051,A -85,B 0,C 180,E1 2222.161,E2 2222.161} C_VEL
LIN {X 0,Y 201.302,Z 514.567,A -85,B 0,C 180,E1 2217.411,E2 2217.411} C_VEL
LIN {X 0,Y 199.352,Z 510.784,A -85,B 0,C 180,E1 2212.881,E2 2212.881} C_VEL
LIN {X 0,Y 197.556,Z 506.897,A -85,B 0,C 180,E1 2206.357,E2 2206.357} C_VEL
LIN {X 0,Y 196.713,Z 506.222,A -85,B 0,C 180,E1 2199.818,E2 2199.818} C_VEL
LIN {X 0,Y 197.361,Z 506.809,A -85,B 0,C 180,E1 2192.763,E2 2192.763} C_VEL
LIN {X 0,Y 197.652,Z 507.435,A -85,B 0,C 180,E1 2191.058,E2 2191.058} C_VEL
LIN {X 0,Y 199.615,Z 511.667,A -85,B 0,C 180,E1 2184.246,E2 2184.246} C_VEL
LIN {X 0,Y 201.863,Z 516.07,A -85,B 0,C 180,E1 2179.377,E2 2179.377} C_VEL
LIN {X 0,Y 204.526,Z 521.265,A -85,B 0,C 180,E1 2174.933,E2 2174.933} C_VEL
LIN {X 0,Y 205.457,Z 523.431,A -85,B 0,C 180,E1 2173.488,E2 2173.488} C_VEL
LIN {X 0,Y 192.724,Z 579.461,A -85,B 0,C 180,E1 2172.817,E2 2172.817} C_VEL
LIN {X 0,Y 185.612,Z 602.889,A -85,B 0,C 180,E1 2172.501,E2 2172.501} C_VEL
LIN {X 0,Y 176.466,Z 626.381,A -85,B 0,C 180,E1 2172.227,E2 2172.227} C_VEL
LIN {X 0,Y 165.873,Z 648.826,A -85,B 0,C 180,E1 2171.821,E2 2171.821} C_VEL
LIN {X 0,Y 154.386,Z 669.347,A -85,B 0,C 180,E1 2171.256,E2 2171.256} C_VEL
LIN {X 0,Y 140.931,Z 689.884,A -85,B 0,C 180,E1 2170.446,E2 2170.446} C_VEL
LIN {X 0,Y 126.39,Z 708.978,A -85,B 0,C 180,E1 2169.356,E2 2169.356} C_VEL
LIN {X 0,Y 111.016,Z 726.472,A -85,B 0,C 180,E1 2167.861,E2 2167.861} C_VEL
LIN {X 0,Y 93.934,Z 743.216,A -85,B 0,C 180,E1 2165.663,E2 2165.663} C_VEL
LIN {X 0,Y 78.069,Z 756.579,A -85,B 0,C 180,E1 2162.771,E2 2162.771} C_VEL
LIN {X 0,Y 60.028,Z 769.747,A -85,B 0,C 180,E1 2157.717,E2 2157.717} C_VEL
LIN {X 0,Y 42.781,Z 780.722,A -85,B 0,C 180,E1 2148.918,E2 2148.918} C_VEL
LIN {X 0,Y 28.31,Z 789.159,A -85,B 0,C 180,E1 2131.956,E2 2131.956} C_VEL
LIN {X 0,Y 19.172,Z 796.356,A -85,B 0,C 180,E1 2090.05,E2 2090.05} C_VEL
LIN {X 0,Y 19.511,Z 798.978,A -85,B 0,C 180,E1 2064.088,E2 2064.088} C_VEL
LIN {X 0,Y 25.128,Z 801.44,A -85,B 0,C 180,E1 2014.579,E2 2014.579} C_VEL
LIN {X 0,Y 17.467,Z 796.066,A -85,B 0,C 180,E1 1973.471,E2 1973.471} C_VEL
LIN {X 0,Y 19.562,Z 790.669,A -85,B 0,C 180,E1 1930.006,E2 1930.006} C_VEL
LIN {X 0,Y 31.374,Z 782.471,A -85,B 0,C 180,E1 1899.076,E2 1899.076} C_VEL
LIN {X 0,Y 48.169,Z 771.872,A -85,B 0,C 180,E1 1884.9,E2 1884.9} C_VEL
LIN {X 0,Y 65.959,Z 759.487,A -85,B 0,C 180,E1 1877.756,E2 1877.756} C_VEL
LIN {X 0,Y 83.983,Z 745.053,A -85,B 0,C 180,E1 1873.405,E2 1873.405} C_VEL
LIN {X 0,Y 100.681,Z 729.595,A -85,B 0,C 180,E1 1870.61,E2 1870.61} C_VEL
LIN {X 0,Y 112.774,Z 717.044,A -85,B 0,C 180,E1 1869.026,E2 1869.026} C_VEL
LIN {X 0,Y 117.589,Z 711.334,A -85,B 0,C 180,E1 1867.977,E2 1867.977} C_VEL
LIN {X 0,Y 128.709,Z 695.345,A -85,B 0,C 180,E1 1864.048,E2 1864.048} C_VEL
LIN {X 0,Y 132.523,Z 689.974,A -85,B 0,C 180,E1 1863.457,E2 1863.457} C_VEL
LIN {X 0,Y 146.824,Z 669.177,A -85,B 0,C 180,E1 1862.58,E2 1862.58} C_VEL
LIN {X 0,Y 159.828,Z 647.006,A -85,B 0,C 180,E1 1861.88,E2 1861.88} C_VEL
LIN {X 0,Y 170.916,Z 624.622,A -85,B 0,C 180,E1 1861.338,E2 1861.338} C_VEL
LIN {X 0,Y 180.516,Z 601.332,A -85,B 0,C 180,E1 1860.901,E2 1860.901} C_VEL
LIN {X 0,Y 188.55,Z 577.277,A -85,B 0,C 180,E1 1860.561,E2 1860.561} C_VEL
LIN {X 0,Y 195.154,Z 551.513,A -85,B 0,C 180,E1 1860.306,E2 1860.306} C_VEL
LIN {X 0,Y 200.895,Z 525.501,A -85,B 0,C 180,E1 1860.067,E2 1860.067} C_VEL
LIN {X 0,Y 198.598,Z 521.038,A -85,B 0,C 180,E1 1855.648,E2 1855.648} C_VEL
